LIN {X 0,Y 408.232,Z 600.263,A -85,B 0,C 180,E1 -11279.744,E2 -11279.744} C_VEL
LIN {X 0,Y 405.316,Z 581.419,A -85,B 0,C 180,E1 -11280.891,E2 -11280.891} C_VEL
LIN {X 0,Y 402.072,Z 568.541,A -85,B 0,C 180,E1 -11281.742,E2 -11281.742} C_VEL
LIN {X 0,Y 400.579,Z 563.488,A -85,B 0,C 180,E1 -11282.113,E2 -11282.113} C_VEL
LIN {X 0,Y 399.742,Z 559.755,A -85,B 0,C 180,E1 -11282.373,E2 -11282.373} C_VEL
LIN {X 0,Y 400.502,Z 548.255,A -85,B 0,C 180,E1 -11285.8,E2 -11285.8} C_VEL
LIN {X 0,Y 401.305,Z 538.061,A -85,B 0,C 180,E1 -11289.085,E2 -11289.085} C_VEL
LIN {X 0,Y 401.725,Z 533.264,A -85,B 0,C 180,E1 -11290.763,E2 -11290.763} C_VEL
LIN {X 0,Y 401.007,Z 527.558,A -85,B 0,C 180,E1 -11293.119,E2 -11293.119} C_VEL
LIN {X 0,Y 400.18,Z 522.98,A -85,B 0,C 180,E1 -11295.374,E2 -11295.374} C_VEL
LIN {X 0,Y 399.225,Z 518.76,A -85,B 0,C 180,E1 -11298.014,E2 -11298.014} C_VEL
LIN {X 0,Y 398.496,Z 515.479,A -85,B 0,C 180,E1 -11300.896,E2 -11300.896} C_VEL
LIN {X 0,Y 398.095,Z 513.82,A -85,B 0,C 180,E1 -11303.114,E2 -11303.114} C_VEL
LIN {X 0,Y 397.825,Z 512.578,A -85,B 0,C 180,E1 -11306.131,E2 -11306.131} C_VEL
LIN {X 0,Y 397.77,Z 512.409,A -85,B 0,C 180,E1 -11308.091,E2 -11308.091} C_VEL
LIN {X 0,Y 399.185,Z 514.86,A -85,B 0,C 180,E1 -11308.431,E2 -11308.431} C_VEL
LIN {X 0,Y 400.849,Z 516.713,A -85,B 0,C 180,E1 -11308.753,E2 -11308.753} C_VEL
LIN {X 0,Y 404.234,Z 521.809,A -85,B 0,C 180,E1 -11309.459,E2 -11309.459} C_VEL
LIN {X 0,Y 409.003,Z 531.362,A -85,B 0,C 180,E1 -11310.53,E2 -11310.53} C_VEL
LIN {X 0,Y 413.279,Z 542.437,A -85,B 0,C 180,E1 -11311.647,E2 -11311.647} C_VEL
LIN {X 0,Y 413.498,Z 543.353,A -85,B 0,C 180,E1 -11311.726,E2 -11311.726} C_VEL
LIN {X 0,Y 411.745,Z 560.994,A -85,B 0,C 180,E1 -11312.784,E2 -11312.784} C_VEL
LIN {X 0,Y 409.989,Z 576.551,A -85,B 0,C 180,E1 -11313.944,E2 -11313.944} C_VEL
LIN {X 0,Y 408.188,Z 591.71,A -85,B 0,C 180,E1 -11315.322,E2 -11315.322} C_VEL
LIN {X 0,Y 406.396,Z 604.533,A -85,B 0,C 180,E1 -11316.703,E2 -11316.703} C_VEL
LIN {X 0,Y 404.87,Z 615.523,A -85,B 0,C 180,E1 -11318.087,E2 -11318.087} C_VEL
LIN {X 0,Y 403.416,Z 625.962,A -85,B 0,C 180,E1 -11319.609,E2 -11319.609} C_VEL
LIN {X 0,Y 401.753,Z 636.685,A -85,B 0,C 180,E1 -11321.445,E2 -11321.445} C_VEL
LIN {X 0,Y 400.536,Z 645.216,A -85,B 0,C 180,E1 -11323.171,E2 -11323.171} C_VEL
LIN {X 0,Y 399.45,Z 652.898,A -85,B 0,C 180,E1 -11324.985,E2 -11324.985} C_VEL
LIN {X 0,Y 398.294,Z 660.864,A -85,B 0,C 180,E1 -11327.258,E2 -11327.258} C_VEL
LIN {X 0,Y 397.602,Z 666.562,A -85,B 0,C 180,E1 -11329.304,E2 -11329.304} C_VEL
LIN {X 0,Y 397.17,Z 670.116,A -85,B 0,C 180,E1 -11330.837,E2 -11330.837} C_VEL
LIN {X 0,Y 396.812,Z 673.807,A -85,B 0,C 180,E1 -11332.879,E2 -11332.879} C_VEL
LIN {X 0,Y 396.486,Z 676.537,A -85,B 0,C 180,E1 -11334.916,E2 -11334.916} C_VEL
LIN {X 0,Y 396.312,Z 678.205,A -85,B 0,C 180,E1 -11336.951,E2 -11336.951} C_VEL
LIN {X 0,Y 396.145,Z 678.944,A -85,B 0,C 180,E1 -11338.984,E2 -11338.984} C_VEL
LIN {X 0,Y 396.116,Z 678.704,A -85,B 0,C 180,E1 -11341.017,E2 -11341.017} C_VEL
LIN {X 0,Y 396.308,Z 677.478,A -85,B 0,C 180,E1 -11343.05,E2 -11343.05} C_VEL
LIN {X 0,Y 396.392,Z 675.323,A -85,B 0,C 180,E1 -11345.086,E2 -11345.086} C_VEL
LIN {X 0,Y 396.634,Z 672.104,A -85,B 0,C 180,E1 -11347.125,E2 -11347.125} C_VEL
LIN {X 0,Y 396.894,Z 667.898,A -85,B 0,C 180,E1 -11349.171,E2 -11349.171} C_VEL
LIN {X 0,Y 397.424,Z 660.965,A -85,B 0,C 180,E1 -11351.734,E2 -11351.734} C_VEL
LIN {X 0,Y 398.273,Z 653.408,A -85,B 0,C 180,E1 -11353.941,E2 -11353.941} C_VEL
LIN {X 0,Y 399.279,Z 644.403,A -85,B 0,C 180,E1 -11356.095,E2 -11356.095} C_VEL
LIN {X 0,Y 400.377,Z 635.474,A -85,B 0,C 180,E1 -11357.89,E2 -11357.89} C_VEL
LIN {X 0,Y 401.652,Z 625.081,A -85,B 0,C 180,E1 -11359.684,E2 -11359.684} C_VEL
LIN {X 0,Y 402.963,Z 614.717,A -85,B 0,C 180,E1 -11361.217,E2 -11361.217} C_VEL
LIN {X 0,Y 404.626,Z 601.75,A -85,B 0,C 180,E1 -11362.851,E2 -11362.851} C_VEL
LIN {X 0,Y 406.197,Z 588.552,A -85,B 0,C 180,E1 -11364.263,E2 -11364.263} C_VEL
LIN {X 0,Y 407.751,Z 574.631,A -85,B 0,C 180,E1 -11365.525,E2 -11365.525} C_VEL
LIN {X 0,Y 409.08,Z 561.456,A -85,B 0,C 180,E1 -11366.531,E2 -11366.531} C_VEL
LIN {X 0,Y 410.589,Z 545.552,A -85,B 0,C 180,E1 -11367.527,E2 -11367.527} C_VEL
LIN {X 0,Y 410.716,Z 541.576,A -85,B 0,C 180,E1 -11367.762,E2 -11367.762} C_VEL
LIN {X 0,Y 404.657,Z 526.643,A -85,B 0,C 180,E1 -11368.967,E2 -11368.967} C_VEL
LIN {X 0,Y 397.755,Z 511.465,A -85,B 0,C 180,E1 -11370.096,E2 -11370.096} C_VEL
LIN {X 0,Y 397.116,Z 509.333,A -85,B 0,C 180,E1 -11370.259,E2 -11370.259} C_VEL
LIN {X 0,Y 397.124,Z 509.331,A -85,B 0,C 180,E1 -11373.718,E2 -11373.718} C_VEL
LIN {X 0,Y 397.102,Z 509.334,A -85,B 0,C 180,E1 -11377.21,E2 -11377.21} C_VEL
LIN {X 0,Y 397.107,Z 509.335,A -85,B 0,C 180,E1 -11380.445,E2 -11380.445} C_VEL
LIN {X 0,Y 397.106,Z 509.333,A -85,B 0,C 180,E1 -11383.648,E2 -11383.648} C_VEL
LIN {X 0,Y 397.108,Z 509.332,A -85,B 0,C 180,E1 -11386.521,E2 -11386.521} C_VEL
LIN {X 0,Y 397.12,Z 509.334,A -85,B 0,C 180,E1 -11390.423,E2 -11390.423} C_VEL
LIN {X 0,Y 397.114,Z 509.336,A -85,B 0,C 180,E1 -11394.265,E2 -11394.265} C_VEL
LIN {X 0,Y 397.12,Z 509.336,A -85,B 0,C 180,E1 -11396.727,E2 -11396.727} C_VEL
LIN {X 0,Y 397.13,Z 509.334,A -85,B 0,C 180,E1 -11400.295,E2 -11400.295} C_VEL
LIN {X 0,Y 397.204,Z 509.363,A -85,B 0,C 180,E1 -11402.466,E2 -11402.466} C_VEL
LIN {X 0,Y 397.787,Z 513.394,A -85,B 0,C 180,E1 -11404.91,E2 -11404.91} C_VEL
LIN {X 0,Y 397.796,Z 518.959,A -85,B 0,C 180,E1 -11408.221,E2 -11408.221} C_VEL
LIN {X 0,Y 397.684,Z 524.314,A -85,B 0,C 180,E1 -11411.451,E2 -11411.451} C_VEL
LIN {X 0,Y 397.658,Z 528.743,A -85,B 0,C 180,E1 -11414.06,E2 -11414.06} C_VEL
LIN {X 0,Y 400.874,Z 536.859,A -85,B 0,C 180,E1 -11414.48,E2 -11414.48} C_VEL
LIN {X 0,Y 407.03,Z 552.39,A -85,B 0,C 180,E1 -11415.394,E2 -11415.394} C_VEL
LIN {X 0,Y 412.436,Z 568.427,A -85,B 0,C 180,E1 -11416.453,E2 -11416.453} C_VEL
LIN {X 0,Y 412.553,Z 570.388,A -85,B 0,C 180,E1 -11416.554,E2 -11416.554} C_VEL
LIN {X 0,Y 411.371,Z 585.54,A -85,B 0,C 180,E1 -11417.32,E2 -11417.32} C_VEL
LIN {X 0,Y 409.951,Z 600.302,A -85,B 0,C 180,E1 -11418.253,E2 -11418.253} C_VEL
LIN {X 0,Y 408.416,Z 614.386,A -85,B 0,C 180,E1 -11419.339,E2 -11419.339} C_VEL
LIN {X 0,Y 406.621,Z 628.646,A -85,B 0,C 180,E1 -11420.674,E2 -11420.674} C_VEL
LIN {X 0,Y 404.874,Z 641.716,A -85,B 0,C 180,E1 -11422.142,E2 -11422.142} C_VEL
LIN {X 0,Y 403.143,Z 653.798,A -85,B 0,C 180,E1 -11423.744,E2 -11423.744} C_VEL
LIN {X 0,Y 401.526,Z 664.929,A -85,B 0,C 180,E1 -11425.481,E2 -11425.481} C_VEL
LIN {X 0,Y 399.981,Z 675.704,A -85,B 0,C 180,E1 -11427.481,E2 -11427.481} C_VEL
LIN {X 0,Y 398.666,Z 684.761,A -85,B 0,C 180,E1 -11429.494,E2 -11429.494} C_VEL
LIN {X 0,Y 398.078,Z 689.301,A -85,B 0,C 180,E1 -11430.665,E2 -11430.665} C_VEL
LIN {X 0,Y 397.078,Z 692.058,A -85,B 0,C 180,E1 -11431.405,E2 -11431.405} C_VEL
LIN {X 0,Y 391.042,Z 699.537,A -85,B 0,C 180,E1 -11433.596,E2 -11433.596} C_VEL
LIN {X 0,Y 389.819,Z 701.752,A -85,B 0,C 180,E1 -11434.383,E2 -11434.383} C_VEL
LIN {X 0,Y 389.682,Z 702.392,A -85,B 0,C 180,E1 -11434.654,E2 -11434.654} C_VEL
LIN {X 0,Y 389.273,Z 706.982,A -85,B 0,C 180,E1 -11436.789,E2 -11436.789} C_VEL
LIN {X 0,Y 389,Z 709.592,A -85,B 0,C 180,E1 -11438.309,E2 -11438.309} C_VEL
LIN {X 0,Y 388.758,Z 712.241,A -85,B 0,C 180,E1 -11440.414,E2 -11440.414} C_VEL
LIN {X 0,Y 388.731,Z 713.972,A -85,B 0,C 180,E1 -11442.529,E2 -11442.529} C_VEL
LIN {X 0,Y 388.595,Z 714.684,A -85,B 0,C 180,E1 -11444.666,E2 -11444.666} C_VEL
LIN {X 0,Y 388.638,Z 714.434,A -85,B 0,C 180,E1 -11446.817,E2 -11446.817} C_VEL
LIN {X 0,Y 388.689,Z 713.166,A -85,B 0,C 180,E1 -11448.992,E2 -11448.992} C_VEL
LIN {X 0,Y 388.909,Z 710.807,A -85,B 0,C 180,E1 -11451.186,E2 -11451.186} C_VEL
LIN {X 0,Y 389.288,Z 707.379,A -85,B 0,C 180,E1 -11453.4,E2 -11453.4} C_VEL
LIN {X 0,Y 389.818,Z 702.644,A -85,B 0,C 180,E1 -11455.65,E2 -11455.65} C_VEL
LIN {X 0,Y 390.549,Z 696.64,A -85,B 0,C 180,E1 -11457.895,E2 -11457.895} C_VEL
LIN {X 0,Y 391.565,Z 689.136,A -85,B 0,C 180,E1 -11460.168,E2 -11460.168} C_VEL
LIN {X 0,Y 392.828,Z 681.236,A -85,B 0,C 180,E1 -11462.156,E2 -11462.156} C_VEL
LIN {X 0,Y 394.372,Z 671.747,A -85,B 0,C 180,E1 -11464.148,E2 -11464.148} C_VEL
LIN {X 0,Y 395.984,Z 662.193,A -85,B 0,C 180,E1 -11465.85,E2 -11465.85} C_VEL
LIN {X 0,Y 397.88,Z 650.516,A -85,B 0,C 180,E1 -11467.631,E2 -11467.631} C_VEL
LIN {X 0,Y 399.917,Z 637.964,A -85,B 0,C 180,E1 -11469.244,E2 -11469.244} C_VEL
LIN {X 0,Y 402.044,Z 623.588,A -85,B 0,C 180,E1 -11470.785,E2 -11470.785} C_VEL
LIN {X 0,Y 404.009,Z 609.267,A -85,B 0,C 180,E1 -11472.044,E2 -11472.044} C_VEL
LIN {X 0,Y 405.508,Z 596.04,A -85,B 0,C 180,E1 -11473.019,E2 -11473.019} C_VEL
LIN {X 0,Y 407.117,Z 580.483,A -85,B 0,C 180,E1 -11473.946,E2 -11473.946} C_VEL
LIN {X 0,Y 407.686,Z 571.505,A -85,B 0,C 180,E1 -11474.403,E2 -11474.403} C_VEL
LIN {X 0,Y 403.383,Z 558.004,A -85,B 0,C 180,E1 -11475.434,E2 -11475.434} C_VEL
LIN {X 0,Y 397.498,Z 543.758,A -85,B 0,C 180,E1 -11476.5,E2 -11476.5} C_VEL
LIN {X 0,Y 392.172,Z 532.891,A -85,B 0,C 180,E1 -11477.32,E2 -11477.32} C_VEL
LIN {X 0,Y 391.082,Z 530.021,A -85,B 0,C 180,E1 -11477.515,E2 -11477.515} C_VEL
LIN {X 0,Y 391.261,Z 524.474,A -85,B 0,C 180,E1 -11481.046,E2 -11481.046} C_VEL
LIN {X 0,Y 391.418,Z 519.979,A -85,B 0,C 180,E1 -11483.897,E2 -11483.897} C_VEL
LIN {X 0,Y 391.231,Z 516.544,A -85,B 0,C 180,E1 -11486.159,E2 -11486.159} C_VEL
LIN {X 0,Y 390.237,Z 511.089,A -85,B 0,C 180,E1 -11489.717,E2 -11489.717} C_VEL
LIN {X 0,Y 390.104,Z 510.207,A -85,B 0,C 180,E1 -11490.358,E2 -11490.358} C_VEL
LIN {X 0,Y 390.106,Z 510.204,A -85,B 0,C 180,E1 -11493.231,E2 -11493.231} C_VEL
LIN {X 0,Y 390.098,Z 510.204,A -85,B 0,C 180,E1 -11496.749,E2 -11496.749} C_VEL
LIN {X 0,Y 390.11,Z 510.207,A -85,B 0,C 180,E1 -11499.983,E2 -11499.983} C_VEL
LIN {X 0,Y 390.128,Z 510.198,A -85,B 0,C 180,E1 -11503.247,E2 -11503.247} C_VEL
LIN {X 0,Y 390.184,Z 510.191,A -85,B 0,C 180,E1 -11506.561,E2 -11506.561} C_VEL
LIN {X 0,Y 390.169,Z 510.193,A -85,B 0,C 180,E1 -11509.622,E2 -11509.622} C_VEL
LIN {X 0,Y 390.309,Z 510.177,A -85,B 0,C 180,E1 -11512.758,E2 -11512.758} C_VEL
LIN {X 0,Y 390.225,Z 510.185,A -85,B 0,C 180,E1 -11514.833,E2 -11514.833} C_VEL
LIN {X 0,Y 390.411,Z 510.161,A -85,B 0,C 180,E1 -11517.936,E2 -11517.936} C_VEL
LIN {X 0,Y 390.541,Z 510.151,A -85,B 0,C 180,E1 -11520,E2 -11520} C_VEL
LIN {X 0,Y 390.307,Z 510.178,A -85,B 0,C 180,E1 -11523.096,E2 -11523.096} C_VEL
LIN {X 0,Y 390.319,Z 510.172,A -85,B 0,C 180,E1 -11526.202,E2 -11526.202} C_VEL
LIN {X 0,Y 390.304,Z 510.174,A -85,B 0,C 180,E1 -11528.282,E2 -11528.282} C_VEL
LIN {X 0,Y 390.168,Z 510.187,A -85,B 0,C 180,E1 -11532.483,E2 -11532.483} C_VEL
LIN {X 0,Y 390.129,Z 510.19,A -85,B 0,C 180,E1 -11535.677,E2 -11535.677} C_VEL
LIN {X 0,Y 390.108,Z 510.177,A -85,B 0,C 180,E1 -11538.921,E2 -11538.921} C_VEL
LIN {X 0,Y 390.1,Z 510.2,A -85,B 0,C 180,E1 -11542.23,E2 -11542.23} C_VEL
LIN {X 0,Y 390.108,Z 510.179,A -85,B 0,C 180,E1 -11545.744,E2 -11545.744} C_VEL
LIN {X 0,Y 390.055,Z 510.213,A -85,B 0,C 180,E1 -11549.109,E2 -11549.109} C_VEL
LIN {X 0,Y 390.034,Z 510.214,A -85,B 0,C 180,E1 -11552.722,E2 -11552.722} C_VEL
LIN {X 0,Y 390.047,Z 510.21,A -85,B 0,C 180,E1 -11555.826,E2 -11555.826} C_VEL
LIN {X 0,Y 390.062,Z 510.224,A -85,B 0,C 180,E1 -11557.06,E2 -11557.06} C_VEL
LIN {X 0,Y 391.812,Z 517.891,A -85,B 0,C 180,E1 -11560.221,E2 -11560.221} C_VEL
LIN {X 0,Y 393.547,Z 526.096,A -85,B 0,C 180,E1 -11563.434,E2 -11563.434} C_VEL
LIN {X 0,Y 395.478,Z 535.006,A -85,B 0,C 180,E1 -11566.769,E2 -11566.769} C_VEL
LIN {X 0,Y 396.313,Z 540.139,A -85,B 0,C 180,E1 -11568.592,E2 -11568.592} C_VEL
LIN {X 0,Y 395.839,Z 547.199,A -85,B 0,C 180,E1 -11570.912,E2 -11570.912} C_VEL
LIN {X 0,Y 394.812,Z 557.025,A -85,B 0,C 180,E1 -11574.027,E2 -11574.027} C_VEL
LIN {X 0,Y 393.841,Z 567.604,A -85,B 0,C 180,E1 -11577.305,E2 -11577.305} C_VEL
LIN {X 0,Y 393.59,Z 570.386,A -85,B 0,C 180,E1 -11578.144,E2 -11578.144} C_VEL
LIN {X 0,Y 399.789,Z 593.013,A -85,B 0,C 180,E1 -11579.311,E2 -11579.311} C_VEL
LIN {X 0,Y 403.572,Z 609.943,A -85,B 0,C 180,E1 -11580.299,E2 -11580.299} C_VEL
LIN {X 0,Y 405.624,Z 620.284,A -85,B 0,C 180,E1 -11580.98,E2 -11580.98} C_VEL
LIN {X 0,Y 404.084,Z 636.161,A -85,B 0,C 180,E1 -11581.859,E2 -11581.859} C_VEL
LIN {X 0,Y 402.301,Z 650.629,A -85,B 0,C 180,E1 -11582.847,E2 -11582.847} C_VEL
LIN {X 0,Y 400.31,Z 665.785,A -85,B 0,C 180,E1 -11584.107,E2 -11584.107} C_VEL
LIN {X 0,Y 398.33,Z 679.819,A -85,B 0,C 180,E1 -11585.506,E2 -11585.506} C_VEL
LIN {X 0,Y 396.467,Z 692.875,A -85,B 0,C 180,E1 -11587.048,E2 -11587.048} C_VEL
LIN {X 0,Y 394.588,Z 705.859,A -85,B 0,C 180,E1 -11588.86,E2 -11588.86} C_VEL
LIN {X 0,Y 393.024,Z 716.9,A -85,B 0,C 180,E1 -11590.683,E2 -11590.683} C_VEL
LIN {X 0,Y 391.815,Z 726.351,A -85,B 0,C 180,E1 -11592.517,E2 -11592.517} C_VEL
LIN {X 0,Y 390.658,Z 735.563,A -85,B 0,C 180,E1 -11594.613,E2 -11594.613} C_VEL
LIN {X 0,Y 389.937,Z 743.324,A -85,B 0,C 180,E1 -11596.72,E2 -11596.72} C_VEL
LIN {X 0,Y 389.28,Z 750.35,A -85,B 0,C 180,E1 -11599.074,E2 -11599.074} C_VEL
LIN {X 0,Y 389.016,Z 755.311,A -85,B 0,C 180,E1 -11601.168,E2 -11601.168} C_VEL
LIN {X 0,Y 388.916,Z 759.796,A -85,B 0,C 180,E1 -11603.66,E2 -11603.66} C_VEL
LIN {X 0,Y 388.73,Z 762.483,A -85,B 0,C 180,E1 -11605.854,E2 -11605.854} C_VEL
LIN {X 0,Y 388.871,Z 763.909,A -85,B 0,C 180,E1 -11607.93,E2 -11607.93} C_VEL
LIN {X 0,Y 388.837,Z 764.362,A -85,B 0,C 180,E1 -11610.001,E2 -11610.001} C_VEL
LIN {X 0,Y 388.937,Z 763.726,A -85,B 0,C 180,E1 -11612.072,E2 -11612.072} C_VEL
LIN {X 0,Y 388.785,Z 762.123,A -85,B 0,C 180,E1 -11614.148,E2 -11614.148} C_VEL
LIN {X 0,Y 388.957,Z 759.368,A -85,B 0,C 180,E1 -11616.395,E2 -11616.395} C_VEL
LIN {X 0,Y 389.029,Z 754.96,A -85,B 0,C 180,E1 -11618.834,E2 -11618.834} C_VEL
LIN {X 0,Y 389.306,Z 750.025,A -85,B 0,C 180,E1 -11620.928,E2 -11620.928} C_VEL
LIN {X 0,Y 389.953,Z 743.004,A -85,B 0,C 180,E1 -11623.29,E2 -11623.29} C_VEL
LIN {X 0,Y 390.796,Z 734.274,A -85,B 0,C 180,E1 -11625.651,E2 -11625.651} C_VEL
LIN {X 0,Y 391.968,Z 724.851,A -85,B 0,C 180,E1 -11627.748,E2 -11627.748} C_VEL
LIN {X 0,Y 393.25,Z 715.147,A -85,B 0,C 180,E1 -11629.579,E2 -11629.579} C_VEL
LIN {X 0,Y 394.82,Z 703.819,A -85,B 0,C 180,E1 -11631.403,E2 -11631.403} C_VEL
LIN {X 0,Y 396.608,Z 691.46,A -85,B 0,C 180,E1 -11633.084,E2 -11633.084} C_VEL
LIN {X 0,Y 398.478,Z 677.931,A -85,B 0,C 180,E1 -11634.626,E2 -11634.626} C_VEL
LIN {X 0,Y 400.243,Z 664.612,A -85,B 0,C 180,E1 -11635.9,E2 -11635.9} C_VEL
LIN {X 0,Y 401.991,Z 650.43,A -85,B 0,C 180,E1 -11637.037,E2 -11637.037} C_VEL
LIN {X 0,Y 403.683,Z 635.143,A -85,B 0,C 180,E1 -11638.039,E2 -11638.039} C_VEL
LIN {X 0,Y 405.114,Z 620.404,A -85,B 0,C 180,E1 -11638.835,E2 -11638.835} C_VEL
LIN {X 0,Y 402.239,Z 602.925,A -85,B 0,C 180,E1 -11640.134,E2 -11640.134} C_VEL
LIN {X 0,Y 399.73,Z 584.771,A -85,B 0,C 180,E1 -11641.317,E2 -11641.317} C_VEL
LIN {X 0,Y 396.715,Z 571.614,A -85,B 0,C 180,E1 -11642.248,E2 -11642.248} C_VEL
LIN {X 0,Y 394.133,Z 562.415,A -85,B 0,C 180,E1 -11642.969,E2 -11642.969} C_VEL
LIN {X 0,Y 393.01,Z 558.534,A -85,B 0,C 180,E1 -11643.296,E2 -11643.296} C_VEL
LIN {X 0,Y 392.946,Z 557.557,A -85,B 0,C 180,E1 -11643.416,E2 -11643.416} C_VEL
LIN {X 0,Y 393.854,Z 546.412,A -85,B 0,C 180,E1 -11646.895,E2 -11646.895} C_VEL
LIN {X 0,Y 394.693,Z 537.205,A -85,B 0,C 180,E1 -11650.034,E2 -11650.034} C_VEL
LIN {X 0,Y 394.715,Z 533.136,A -85,B 0,C 180,E1 -11651.599,E2 -11651.599} C_VEL
LIN {X 0,Y 393.875,Z 527.61,A -85,B 0,C 180,E1 -11654.099,E2 -11654.099} C_VEL
LIN {X 0,Y 393.042,Z 523.275,A -85,B 0,C 180,E1 -11656.495,E2 -11656.495} C_VEL
LIN {X 0,Y 392.021,Z 518.861,A -85,B 0,C 180,E1 -11659.805,E2 -11659.805} C_VEL
LIN {X 0,Y 391.498,Z 516.574,A -85,B 0,C 180,E1 -11662.385,E2 -11662.385} C_VEL
LIN {X 0,Y 391.099,Z 514.905,A -85,B 0,C 180,E1 -11665.753,E2 -11665.753} C_VEL
LIN {X 0,Y 391.038,Z 514.772,A -85,B 0,C 180,E1 -11667.127,E2 -11667.127} C_VEL
LIN {X 0,Y 392.595,Z 517.244,A -85,B 0,C 180,E1 -11667.534,E2 -11667.534} C_VEL
LIN {X 0,Y 394.151,Z 518.801,A -85,B 0,C 180,E1 -11667.87,E2 -11667.87} C_VEL
LIN {X 0,Y 398.297,Z 524.304,A -85,B 0,C 180,E1 -11668.787,E2 -11668.787} C_VEL
LIN {X 0,Y 403.505,Z 534.578,A -85,B 0,C 180,E1 -11670.061,E2 -11670.061} C_VEL
LIN {X 0,Y 407.507,Z 545.247,A -85,B 0,C 180,E1 -11671.204,E2 -11671.204} C_VEL
LIN {X 0,Y 405.829,Z 562.036,A -85,B 0,C 180,E1 -11672.253,E2 -11672.253} C_VEL
LIN {X 0,Y 404.001,Z 576.936,A -85,B 0,C 180,E1 -11673.388,E2 -11673.388} C_VEL
LIN {X 0,Y 402.224,Z 590.843,A -85,B 0,C 180,E1 -11674.654,E2 -11674.654} C_VEL
LIN {X 0,Y 400.211,Z 604.901,A -85,B 0,C 180,E1 -11676.178,E2 -11676.178} C_VEL
LIN {X 0,Y 398.428,Z 616.898,A -85,B 0,C 180,E1 -11677.714,E2 -11677.714} C_VEL
LIN {X 0,Y 396.631,Z 628.788,A -85,B 0,C 180,E1 -11679.516,E2 -11679.516} C_VEL
LIN {X 0,Y 394.961,Z 638.951,A -85,B 0,C 180,E1 -11681.32,E2 -11681.32} C_VEL
LIN {X 0,Y 393.416,Z 648.664,A -85,B 0,C 180,E1 -11683.392,E2 -11683.392} C_VEL
LIN {X 0,Y 392.233,Z 656.733,A -85,B 0,C 180,E1 -11685.473,E2 -11685.473} C_VEL
LIN {X 0,Y 391.201,Z 663.389,A -85,B 0,C 180,E1 -11687.551,E2 -11687.551} C_VEL
LIN {X 0,Y 390.582,Z 668.818,A -85,B 0,C 180,E1 -11689.634,E2 -11689.634} C_VEL
LIN {X 0,Y 390.038,Z 673.053,A -85,B 0,C 180,E1 -11691.712,E2 -11691.712} C_VEL
LIN {X 0,Y 389.722,Z 676.204,A -85,B 0,C 180,E1 -11693.789,E2 -11693.789} C_VEL
LIN {X 0,Y 389.446,Z 678.388,A -85,B 0,C 180,E1 -11695.861,E2 -11695.861} C_VEL
LIN {X 0,Y 389.175,Z 679.546,A -85,B 0,C 180,E1 -11697.931,E2 -11697.931} C_VEL
LIN {X 0,Y 389.059,Z 679.802,A -85,B 0,C 180,E1 -11700,E2 -11700} C_VEL
LIN {X 0,Y 389.136,Z 678.995,A -85,B 0,C 180,E1 -11702.07,E2 -11702.07} C_VEL
LIN {X 0,Y 389.385,Z 677.273,A -85,B 0,C 180,E1 -11704.141,E2 -11704.141} C_VEL
LIN {X 0,Y 389.351,Z 674.549,A -85,B 0,C 180,E1 -11706.218,E2 -11706.218} C_VEL
LIN {X 0,Y 389.706,Z 670.773,A -85,B 0,C 180,E1 -11708.296,E2 -11708.296} C_VEL
LIN {X 0,Y 390.054,Z 665.928,A -85,B 0,C 180,E1 -11710.381,E2 -11710.381} C_VEL
LIN {X 0,Y 390.629,Z 659.834,A -85,B 0,C 180,E1 -11712.469,E2 -11712.469} C_VEL
LIN {X 0,Y 391.46,Z 652.448,A -85,B 0,C 180,E1 -11714.558,E2 -11714.558} C_VEL
LIN {X 0,Y 392.597,Z 643.583,A -85,B 0,C 180,E1 -11716.644,E2 -11716.644} C_VEL
LIN {X 0,Y 393.969,Z 632.977,A -85,B 0,C 180,E1 -11718.73,E2 -11718.73} C_VEL
LIN {X 0,Y 395.351,Z 621.954,A -85,B 0,C 180,E1 -11720.554,E2 -11720.554} C_VEL
LIN {X 0,Y 396.836,Z 610.953,A -85,B 0,C 180,E1 -11722.108,E2 -11722.108} C_VEL
LIN {X 0,Y 398.342,Z 599.269,A -85,B 0,C 180,E1 -11723.541,E2 -11723.541} C_VEL
LIN {X 0,Y 400.158,Z 584.503,A -85,B 0,C 180,E1 -11725.069,E2 -11725.069} C_VEL
LIN {X 0,Y 401.723,Z 571.203,A -85,B 0,C 180,E1 -11726.215,E2 -11726.215} C_VEL
LIN {X 0,Y 403.139,Z 556.268,A -85,B 0,C 180,E1 -11727.307,E2 -11727.307} C_VEL
LIN {X 0,Y 404.236,Z 543.771,A -85,B 0,C 180,E1 -11728.073,E2 -11728.073} C_VEL
LIN {X 0,Y 397.518,Z 527.206,A -85,B 0,C 180,E1 -11729.456,E2 -11729.456} C_VEL
LIN {X 0,Y 390.79,Z 512.6,A -85,B 0,C 180,E1 -11730.573,E2 -11730.573} C_VEL
LIN {X 0,Y 390.062,Z 510.212,A -85,B 0,C 180,E1 -11730.732,E2 -11730.732} C_VEL
LIN {X 0,Y 390.073,Z 510.209,A -85,B 0,C 180,E1 -11734.025,E2 -11734.025} C_VEL
LIN {X 0,Y 390.05,Z 510.214,A -85,B 0,C 180,E1 -11737.551,E2 -11737.551} C_VEL
LIN {X 0,Y 390.061,Z 510.211,A -85,B 0,C 180,E1 -11740.821,E2 -11740.821} C_VEL
LIN {X 0,Y 390.06,Z 510.21,A -85,B 0,C 180,E1 -11743.886,E2 -11743.886} C_VEL
LIN {X 0,Y 390.063,Z 510.209,A -85,B 0,C 180,E1 -11746.79,E2 -11746.79} C_VEL
LIN {X 0,Y 390.062,Z 510.21,A -85,B 0,C 180,E1 -11749.56,E2 -11749.56} C_VEL
LIN {X 0,Y 390.049,Z 510.212,A -85,B 0,C 180,E1 -11752.449,E2 -11752.449} C_VEL
LIN {X 0,Y 390.074,Z 510.214,A -85,B 0,C 180,E1 -11756.045,E2 -11756.045} C_VEL
LIN {X 0,Y 390.053,Z 510.217,A -85,B 0,C 180,E1 -11759.869,E2 -11759.869} C_VEL
LIN {X 0,Y 390.157,Z 510.377,A -85,B 0,C 180,E1 -11762.218,E2 -11762.218} C_VEL
LIN {X 0,Y 390.754,Z 514.002,A -85,B 0,C 180,E1 -11764.426,E2 -11764.426} C_VEL
LIN {X 0,Y 390.847,Z 517.77,A -85,B 0,C 180,E1 -11766.696,E2 -11766.696} C_VEL
LIN {X 0,Y 390.769,Z 523.277,A -85,B 0,C 180,E1 -11770.018,E2 -11770.018} C_VEL
LIN {X 0,Y 390.674,Z 528.948,A -85,B 0,C 180,E1 -11773.482,E2 -11773.482} C_VEL
LIN {X 0,Y 391.754,Z 532.057,A -85,B 0,C 180,E1 -11773.655,E2 -11773.655} C_VEL
LIN {X 0,Y 399.059,Z 549.937,A -85,B 0,C 180,E1 -11774.705,E2 -11774.705} C_VEL
LIN {X 0,Y 404.447,Z 565.332,A -85,B 0,C 180,E1 -11775.715,E2 -11775.715} C_VEL
LIN {X 0,Y 406.187,Z 571.314,A -85,B 0,C 180,E1 -11776.133,E2 -11776.133} C_VEL
LIN {X 0,Y 404.884,Z 587.171,A -85,B 0,C 180,E1 -11776.958,E2 -11776.958} C_VEL
LIN {X 0,Y 403.362,Z 602.056,A -85,B 0,C 180,E1 -11777.93,E2 -11777.93} C_VEL
LIN {X 0,Y 401.781,Z 615.905,A -85,B 0,C 180,E1 -11779.033,E2 -11779.033} C_VEL
LIN {X 0,Y 399.952,Z 630.054,A -85,B 0,C 180,E1 -11780.389,E2 -11780.389} C_VEL
LIN {X 0,Y 398.132,Z 642.987,A -85,B 0,C 180,E1 -11781.881,E2 -11781.881} C_VEL
LIN {X 0,Y 396.454,Z 654.101,A -85,B 0,C 180,E1 -11783.382,E2 -11783.382} C_VEL
LIN {X 0,Y 394.788,Z 665.26,A -85,B 0,C 180,E1 -11785.148,E2 -11785.148} C_VEL
LIN {X 0,Y 393.165,Z 676.055,A -85,B 0,C 180,E1 -11787.181,E2 -11787.181} C_VEL
LIN {X 0,Y 391.764,Z 685.127,A -85,B 0,C 180,E1 -11789.228,E2 -11789.228} C_VEL
LIN {X 0,Y 390.864,Z 691.831,A -85,B 0,C 180,E1 -11791.029,E2 -11791.029} C_VEL
LIN {X 0,Y 390.031,Z 698.359,A -85,B 0,C 180,E1 -11793.098,E2 -11793.098} C_VEL
LIN {X 0,Y 389.682,Z 702.392,A -85,B 0,C 180,E1 -11794.654,E2 -11794.654} C_VEL
LIN {X 0,Y 388.855,Z 704.361,A -85,B 0,C 180,E1 -11795.464,E2 -11795.464} C_VEL
LIN {X 0,Y 385.718,Z 707.32,A -85,B 0,C 180,E1 -11796.786,E2 -11796.786} C_VEL
LIN {X 0,Y 383.095,Z 709.374,A -85,B 0,C 180,E1 -11797.868,E2 -11797.868} C_VEL
LIN {X 0,Y 381.931,Z 710.719,A -85,B 0,C 180,E1 -11798.718,E2 -11798.718} C_VEL
LIN {X 0,Y 381.813,Z 711.109,A -85,B 0,C 180,E1 -11799.009,E2 -11799.009} C_VEL
LIN {X 0,Y 381.676,Z 712.948,A -85,B 0,C 180,E1 -11800.609,E2 -11800.609} C_VEL
LIN {X 0,Y 381.611,Z 714.536,A -85,B 0,C 180,E1 -11802.766,E2 -11802.766} C_VEL
LIN {X 0,Y 381.506,Z 715.177,A -85,B 0,C 180,E1 -11804.944,E2 -11804.944} C_VEL
LIN {X 0,Y 381.567,Z 714.778,A -85,B 0,C 180,E1 -11807.138,E2 -11807.138} C_VEL
LIN {X 0,Y 381.645,Z 713.429,A -85,B 0,C 180,E1 -11809.357,E2 -11809.357} C_VEL
LIN {X 0,Y 381.905,Z 710.921,A -85,B 0,C 180,E1 -11811.594,E2 -11811.594} C_VEL
LIN {X 0,Y 382.338,Z 707.326,A -85,B 0,C 180,E1 -11813.852,E2 -11813.852} C_VEL
LIN {X 0,Y 382.951,Z 702.535,A -85,B 0,C 180,E1 -11816.131,E2 -11816.131} C_VEL
LIN {X 0,Y 383.775,Z 696.205,A -85,B 0,C 180,E1 -11818.475,E2 -11818.475} C_VEL
LIN {X 0,Y 385.025,Z 688.006,A -85,B 0,C 180,E1 -11820.917,E2 -11820.917} C_VEL
LIN {X 0,Y 386.488,Z 679.215,A -85,B 0,C 180,E1 -11823.059,E2 -11823.059} C_VEL
LIN {X 0,Y 388.212,Z 669.304,A -85,B 0,C 180,E1 -11825.083,E2 -11825.083} C_VEL
LIN {X 0,Y 390.038,Z 659.373,A -85,B 0,C 180,E1 -11826.805,E2 -11826.805} C_VEL
LIN {X 0,Y 391.965,Z 647.61,A -85,B 0,C 180,E1 -11828.539,E2 -11828.539} C_VEL
LIN {X 0,Y 394.099,Z 634.952,A -85,B 0,C 180,E1 -11830.105,E2 -11830.105} C_VEL
LIN {X 0,Y 396.199,Z 621.076,A -85,B 0,C 180,E1 -11831.551,E2 -11831.551} C_VEL
LIN {X 0,Y 398.209,Z 606.559,A -85,B 0,C 180,E1 -11832.801,E2 -11832.801} C_VEL
LIN {X 0,Y 399.985,Z 591.759,A -85,B 0,C 180,E1 -11833.847,E2 -11833.847} C_VEL
LIN {X 0,Y 401.508,Z 576.128,A -85,B 0,C 180,E1 -11834.721,E2 -11834.721} C_VEL
LIN {X 0,Y 401.648,Z 574.562,A -85,B 0,C 180,E1 -11834.802,E2 -11834.802} C_VEL
LIN {X 0,Y 399.455,Z 566.295,A -85,B 0,C 180,E1 -11835.444,E2 -11835.444} C_VEL
LIN {X 0,Y 394.724,Z 553.39,A -85,B 0,C 180,E1 -11836.462,E2 -11836.462} C_VEL
LIN {X 0,Y 388.951,Z 540.503,A -85,B 0,C 180,E1 -11837.479,E2 -11837.479} C_VEL
LIN {X 0,Y 384.469,Z 531.49,A -85,B 0,C 180,E1 -11838.182,E2 -11838.182} C_VEL
LIN {X 0,Y 384.212,Z 530.464,A -85,B 0,C 180,E1 -11838.259,E2 -11838.259} C_VEL
LIN {X 0,Y 384.41,Z 524.912,A -85,B 0,C 180,E1 -11841.824,E2 -11841.824} C_VEL
LIN {X 0,Y 384.504,Z 521.219,A -85,B 0,C 180,E1 -11844.204,E2 -11844.204} C_VEL
LIN {X 0,Y 384.447,Z 519.277,A -85,B 0,C 180,E1 -11845.479,E2 -11845.479} C_VEL
LIN {X 0,Y 383.9,Z 515.687,A -85,B 0,C 180,E1 -11847.933,E2 -11847.933} C_VEL
LIN {X 0,Y 383.029,Z 511.09,A -85,B 0,C 180,E1 -11850.981,E2 -11850.981} C_VEL
LIN {X 0,Y 383.072,Z 511.083,A -85,B 0,C 180,E1 -11854.02,E2 -11854.02} C_VEL
LIN {X 0,Y 383.005,Z 511.09,A -85,B 0,C 180,E1 -11857.334,E2 -11857.334} C_VEL
LIN {X 0,Y 383.063,Z 511.08,A -85,B 0,C 180,E1 -11860.716,E2 -11860.716} C_VEL
LIN {X 0,Y 383.071,Z 511.078,A -85,B 0,C 180,E1 -11864.026,E2 -11864.026} C_VEL
LIN {X 0,Y 383.131,Z 511.075,A -85,B 0,C 180,E1 -11867.283,E2 -11867.283} C_VEL
LIN {X 0,Y 383.147,Z 511.073,A -85,B 0,C 180,E1 -11870.497,E2 -11870.497} C_VEL
LIN {X 0,Y 383.264,Z 511.053,A -85,B 0,C 180,E1 -11872.625,E2 -11872.625} C_VEL
LIN {X 0,Y 383.197,Z 511.06,A -85,B 0,C 180,E1 -11874.738,E2 -11874.738} C_VEL
LIN {X 0,Y 383.378,Z 511.037,A -85,B 0,C 180,E1 -11877.898,E2 -11877.898} C_VEL
LIN {X 0,Y 383.511,Z 511.027,A -85,B 0,C 180,E1 -11880,E2 -11880} C_VEL
LIN {X 0,Y 383.243,Z 511.058,A -85,B 0,C 180,E1 -11883.153,E2 -11883.153} C_VEL
LIN {X 0,Y 383.276,Z 511.05,A -85,B 0,C 180,E1 -11886.316,E2 -11886.316} C_VEL
LIN {X 0,Y 383.249,Z 511.051,A -85,B 0,C 180,E1 -11888.435,E2 -11888.435} C_VEL
LIN {X 0,Y 383.098,Z 511.071,A -85,B 0,C 180,E1 -11891.642,E2 -11891.642} C_VEL
LIN {X 0,Y 383.101,Z 511.075,A -85,B 0,C 180,E1 -11894.882,E2 -11894.882} C_VEL
LIN {X 0,Y 383.083,Z 511.041,A -85,B 0,C 180,E1 -11898.172,E2 -11898.172} C_VEL
LIN {X 0,Y 383.063,Z 511.082,A -85,B 0,C 180,E1 -11901.526,E2 -11901.526} C_VEL
LIN {X 0,Y 383.043,Z 511.049,A -85,B 0,C 180,E1 -11904.96,E2 -11904.96} C_VEL
LIN {X 0,Y 383.039,Z 511.085,A -85,B 0,C 180,E1 -11908.492,E2 -11908.492} C_VEL
LIN {X 0,Y 383.002,Z 511.089,A -85,B 0,C 180,E1 -11912.15,E2 -11912.15} C_VEL
LIN {X 0,Y 383.008,Z 511.087,A -85,B 0,C 180,E1 -11914.668,E2 -11914.668} C_VEL
LIN {X 0,Y 383.038,Z 511.132,A -85,B 0,C 180,E1 -11916.513,E2 -11916.513} C_VEL
LIN {X 0,Y 384.853,Z 519.24,A -85,B 0,C 180,E1 -11919.919,E2 -11919.919} C_VEL
LIN {X 0,Y 386.701,Z 527.921,A -85,B 0,C 180,E1 -11923.369,E2 -11923.369} C_VEL
LIN {X 0,Y 388.816,Z 537.742,A -85,B 0,C 180,E1 -11927.088,E2 -11927.088} C_VEL
LIN {X 0,Y 389.415,Z 542.483,A -85,B 0,C 180,E1 -11928.778,E2 -11928.778} C_VEL
LIN {X 0,Y 388.642,Z 550.81,A -85,B 0,C 180,E1 -11931.523,E2 -11931.523} C_VEL
LIN {X 0,Y 387.667,Z 560.619,A -85,B 0,C 180,E1 -11934.666,E2 -11934.666} C_VEL
LIN {X 0,Y 386.807,Z 569.997,A -85,B 0,C 180,E1 -11937.551,E2 -11937.551} C_VEL
LIN {X 0,Y 393.339,Z 593.753,A -85,B 0,C 180,E1 -11938.829,E2 -11938.829} C_VEL
LIN {X 0,Y 396.924,Z 610.361,A -85,B 0,C 180,E1 -11939.828,E2 -11939.828} C_VEL
LIN {X 0,Y 399.148,Z 621.796,A -85,B 0,C 180,E1 -11940.611,E2 -11940.611} C_VEL
LIN {X 0,Y 397.296,Z 638.989,A -85,B 0,C 180,E1 -11941.616,E2 -11941.616} C_VEL
LIN {X 0,Y 395.159,Z 654.932,A -85,B 0,C 180,E1 -11942.78,E2 -11942.78} C_VEL
LIN {X 0,Y 393.013,Z 670.376,A -85,B 0,C 180,E1 -11944.16,E2 -11944.16} C_VEL
LIN {X 0,Y 391.125,Z 683.732,A -85,B 0,C 180,E1 -11945.59,E2 -11945.59} C_VEL
LIN {X 0,Y 389.16,Z 696.344,A -85,B 0,C 180,E1 -11947.184,E2 -11947.184} C_VEL
LIN {X 0,Y 387.301,Z 708.441,A -85,B 0,C 180,E1 -11949,E2 -11949} C_VEL
LIN {X 0,Y 385.638,Z 720.05,A -85,B 0,C 180,E1 -11951.069,E2 -11951.069} C_VEL
LIN {X 0,Y 384.46,Z 729.291,A -85,B 0,C 180,E1 -11952.995,E2 -11952.995} C_VEL
LIN {X 0,Y 383.34,Z 737.904,A -85,B 0,C 180,E1 -11955.129,E2 -11955.129} C_VEL
LIN {X 0,Y 382.659,Z 745.088,A -85,B 0,C 180,E1 -11957.269,E2 -11957.269} C_VEL
LIN {X 0,Y 382.091,Z 750.979,A -85,B 0,C 180,E1 -11959.402,E2 -11959.402} C_VEL
LIN {X 0,Y 381.89,Z 755.699,A -85,B 0,C 180,E1 -11961.535,E2 -11961.535} C_VEL
LIN {X 0,Y 381.844,Z 759.255,A -85,B 0,C 180,E1 -11963.661,E2 -11963.661} C_VEL
LIN {X 0,Y 381.661,Z 761.773,A -85,B 0,C 180,E1 -11965.777,E2 -11965.777} C_VEL
LIN {X 0,Y 381.802,Z 763.188,A -85,B 0,C 180,E1 -11967.891,E2 -11967.891} C_VEL
LIN {X 0,Y 381.793,Z 763.675,A -85,B 0,C 180,E1 -11970.001,E2 -11970.001} C_VEL
LIN {X 0,Y 381.863,Z 763.145,A -85,B 0,C 180,E1 -11972.111,E2 -11972.111} C_VEL
LIN {X 0,Y 381.708,Z 761.69,A -85,B 0,C 180,E1 -11974.225,E2 -11974.225} C_VEL
LIN {X 0,Y 381.885,Z 759.066,A -85,B 0,C 180,E1 -11976.394,E2 -11976.394} C_VEL
LIN {X 0,Y 381.934,Z 754.496,A -85,B 0,C 180,E1 -11979,E2 -11979} C_VEL
LIN {X 0,Y 382.27,Z 749.561,A -85,B 0,C 180,E1 -11981.131,E2 -11981.131} C_VEL
LIN {X 0,Y 382.878,Z 743.02,A -85,B 0,C 180,E1 -11983.383,E2 -11983.383} C_VEL
LIN {X 0,Y 383.713,Z 734.831,A -85,B 0,C 180,E1 -11985.675,E2 -11985.675} C_VEL
LIN {X 0,Y 384.899,Z 725.61,A -85,B 0,C 180,E1 -11987.81,E2 -11987.81} C_VEL
LIN {X 0,Y 386.437,Z 714.617,A -85,B 0,C 180,E1 -11989.939,E2 -11989.939} C_VEL
LIN {X 0,Y 388.086,Z 703.252,A -85,B 0,C 180,E1 -11991.793,E2 -11991.793} C_VEL
LIN {X 0,Y 389.964,Z 690.88,A -85,B 0,C 180,E1 -11993.5,E2 -11993.5} C_VEL
LIN {X 0,Y 391.908,Z 677.333,A -85,B 0,C 180,E1 -11995.067,E2 -11995.067} C_VEL
LIN {X 0,Y 393.788,Z 663.969,A -85,B 0,C 180,E1 -11996.357,E2 -11996.357} C_VEL
LIN {X 0,Y 395.585,Z 649.701,A -85,B 0,C 180,E1 -11997.512,E2 -11997.512} C_VEL
LIN {X 0,Y 397.379,Z 634.32,A -85,B 0,C 180,E1 -11998.524,E2 -11998.524} C_VEL
LIN {X 0,Y 398.671,Z 622.184,A -85,B 0,C 180,E1 -11999.23,E2 -11999.23} C_VEL
LIN {X 0,Y 396.234,Z 605.191,A -85,B 0,C 180,E1 -12000.566,E2 -12000.566} C_VEL
LIN {X 0,Y 393.942,Z 586.52,A -85,B 0,C 180,E1 -12001.873,E2 -12001.873} C_VEL
LIN {X 0,Y 390.732,Z 571.653,A -85,B 0,C 180,E1 -12003.003,E2 -12003.003} C_VEL
LIN {X 0,Y 387.51,Z 560.649,A -85,B 0,C 180,E1 -12003.985,E2 -12003.985} C_VEL
LIN {X 0,Y 386.257,Z 556.104,A -85,B 0,C 180,E1 -12004.408,E2 -12004.408} C_VEL
LIN {X 0,Y 386.225,Z 555.424,A -85,B 0,C 180,E1 -12004.522,E2 -12004.522} C_VEL
LIN {X 0,Y 387.022,Z 546.395,A -85,B 0,C 180,E1 -12007.469,E2 -12007.469} C_VEL
LIN {X 0,Y 387.967,Z 537.351,A -85,B 0,C 180,E1 -12010.704,E2 -12010.704} C_VEL
LIN {X 0,Y 387.549,Z 532.442,A -85,B 0,C 180,E1 -12012.798,E2 -12012.798} C_VEL
LIN {X 0,Y 386.788,Z 527.839,A -85,B 0,C 180,E1 -12015.125,E2 -12015.125} C_VEL
LIN {X 0,Y 385.882,Z 523.863,A -85,B 0,C 180,E1 -12017.634,E2 -12017.634} C_VEL
LIN {X 0,Y 385.198,Z 520.649,A -85,B 0,C 180,E1 -12020.315,E2 -12020.315} C_VEL
LIN {X 0,Y 384.603,Z 518.154,A -85,B 0,C 180,E1 -12023.518,E2 -12023.518} C_VEL
LIN {X 0,Y 384.367,Z 517.124,A -85,B 0,C 180,E1 -12026.016,E2 -12026.016} C_VEL
LIN {X 0,Y 385.911,Z 519.589,A -85,B 0,C 180,E1 -12026.486,E2 -12026.486} C_VEL
LIN {X 0,Y 387.632,Z 521.236,A -85,B 0,C 180,E1 -12026.913,E2 -12026.913} C_VEL
LIN {X 0,Y 389.925,Z 523.96,A -85,B 0,C 180,E1 -12027.482,E2 -12027.482} C_VEL
LIN {X 0,Y 394.307,Z 530.118,A -85,B 0,C 180,E1 -12028.548,E2 -12028.548} C_VEL
LIN {X 0,Y 399.22,Z 540.739,A -85,B 0,C 180,E1 -12029.904,E2 -12029.904} C_VEL
LIN {X 0,Y 401.546,Z 547.353,A -85,B 0,C 180,E1 -12030.656,E2 -12030.656} C_VEL
LIN {X 0,Y 401.721,Z 549.089,A -85,B 0,C 180,E1 -12030.793,E2 -12030.793} C_VEL
LIN {X 0,Y 399.862,Z 564.617,A -85,B 0,C 180,E1 -12031.802,E2 -12031.802} C_VEL
LIN {X 0,Y 397.754,Z 580.646,A -85,B 0,C 180,E1 -12033.079,E2 -12033.079} C_VEL
LIN {X 0,Y 395.71,Z 595.179,A -85,B 0,C 180,E1 -12034.489,E2 -12034.489} C_VEL
LIN {X 0,Y 393.605,Z 608.68,A -85,B 0,C 180,E1 -12036.033,E2 -12036.033} C_VEL
LIN {X 0,Y 391.744,Z 620.142,A -85,B 0,C 180,E1 -12037.591,E2 -12037.591} C_VEL
LIN {X 0,Y 389.828,Z 631.659,A -85,B 0,C 180,E1 -12039.419,E2 -12039.419} C_VEL
LIN {X 0,Y 388.129,Z 641.457,A -85,B 0,C 180,E1 -12041.252,E2 -12041.252} C_VEL
LIN {X 0,Y 386.714,Z 649.855,A -85,B 0,C 180,E1 -12043.096,E2 -12043.096} C_VEL
LIN {X 0,Y 385.433,Z 657.835,A -85,B 0,C 180,E1 -12045.211,E2 -12045.211} C_VEL
LIN {X 0,Y 384.35,Z 664.467,A -85,B 0,C 180,E1 -12047.325,E2 -12047.325} C_VEL
LIN {X 0,Y 383.656,Z 669.835,A -85,B 0,C 180,E1 -12049.445,E2 -12049.445} C_VEL
LIN {X 0,Y 383.077,Z 674.028,A -85,B 0,C 180,E1 -12051.561,E2 -12051.561} C_VEL
LIN {X 0,Y 382.723,Z 677.153,A -85,B 0,C 180,E1 -12053.675,E2 -12053.675} C_VEL
LIN {X 0,Y 382.424,Z 679.305,A -85,B 0,C 180,E1 -12055.785,E2 -12055.785} C_VEL
LIN {X 0,Y 382.132,Z 680.415,A -85,B 0,C 180,E1 -12057.892,E2 -12057.892} C_VEL
LIN {X 0,Y 382.008,Z 680.629,A -85,B 0,C 180,E1 -12060,E2 -12060} C_VEL
LIN {X 0,Y 382.093,Z 679.776,A -85,B 0,C 180,E1 -12062.109,E2 -12062.109} C_VEL
LIN {X 0,Y 382.328,Z 678.013,A -85,B 0,C 180,E1 -12064.217,E2 -12064.217} C_VEL
LIN {X 0,Y 382.323,Z 675.238,A -85,B 0,C 180,E1 -12066.333,E2 -12066.333} C_VEL
LIN {X 0,Y 382.697,Z 671.41,A -85,B 0,C 180,E1 -12068.449,E2 -12068.449} C_VEL
LIN {X 0,Y 383.075,Z 666.51,A -85,B 0,C 180,E1 -12070.572,E2 -12070.572} C_VEL
LIN {X 0,Y 383.698,Z 660.34,A -85,B 0,C 180,E1 -12072.698,E2 -12072.698} C_VEL
LIN {X 0,Y 384.552,Z 652.882,A -85,B 0,C 180,E1 -12074.825,E2 -12074.825} C_VEL
LIN {X 0,Y 385.76,Z 643.922,A -85,B 0,C 180,E1 -12076.948,E2 -12076.948} C_VEL
LIN {X 0,Y 387.191,Z 633.217,A -85,B 0,C 180,E1 -12079.07,E2 -12079.07} C_VEL
LIN {X 0,Y 388.641,Z 622.124,A -85,B 0,C 180,E1 -12080.926,E2 -12080.926} C_VEL
LIN {X 0,Y 390.176,Z 611.011,A -85,B 0,C 180,E1 -12082.505,E2 -12082.505} C_VEL
LIN {X 0,Y 392.053,Z 597.154,A -85,B 0,C 180,E1 -12084.186,E2 -12084.186} C_VEL
LIN {X 0,Y 393.799,Z 582.864,A -85,B 0,C 180,E1 -12085.645,E2 -12085.645} C_VEL
LIN {X 0,Y 395.467,Z 569.523,A -85,B 0,C 180,E1 -12086.788,E2 -12086.788} C_VEL
LIN {X 0,Y 396.628,Z 557.128,A -85,B 0,C 180,E1 -12087.693,E2 -12087.693} C_VEL
LIN {X 0,Y 397.696,Z 545.879,A -85,B 0,C 180,E1 -12088.396,E2 -12088.396} C_VEL
LIN {X 0,Y 391.908,Z 531.419,A -85,B 0,C 180,E1 -12089.65,E2 -12089.65} C_VEL
LIN {X 0,Y 384.202,Z 514.226,A -85,B 0,C 180,E1 -12091.013,E2 -12091.013} C_VEL
LIN {X 0,Y 383.067,Z 511.603,A -85,B 0,C 180,E1 -12091.206,E2 -12091.206} C_VEL
LIN {X 0,Y 383.003,Z 511.091,A -85,B 0,C 180,E1 -12091.248,E2 -12091.248} C_VEL
LIN {X 0,Y 383.023,Z 511.09,A -85,B 0,C 180,E1 -12094.668,E2 -12094.668} C_VEL
LIN {X 0,Y 383.006,Z 511.089,A -85,B 0,C 180,E1 -12097.904,E2 -12097.904} C_VEL
LIN {X 0,Y 382.989,Z 511.092,A -85,B 0,C 180,E1 -12101.347,E2 -12101.347} C_VEL
LIN {X 0,Y 383.001,Z 511.091,A -85,B 0,C 180,E1 -12104.303,E2 -12104.303} C_VEL
LIN {X 0,Y 383.016,Z 511.088,A -85,B 0,C 180,E1 -12107.24,E2 -12107.24} C_VEL
LIN {X 0,Y 383.021,Z 511.09,A -85,B 0,C 180,E1 -12110.413,E2 -12110.413} C_VEL
LIN {X 0,Y 383.031,Z 511.09,A -85,B 0,C 180,E1 -12114.044,E2 -12114.044} C_VEL
LIN {X 0,Y 382.993,Z 511.095,A -85,B 0,C 180,E1 -12117.578,E2 -12117.578} C_VEL
LIN {X 0,Y 382.998,Z 511.094,A -85,B 0,C 180,E1 -12120.3,E2 -12120.3} C_VEL
LIN {X 0,Y 383.08,Z 511.224,A -85,B 0,C 180,E1 -12121.831,E2 -12121.831} C_VEL
LIN {X 0,Y 383.66,Z 514.604,A -85,B 0,C 180,E1 -12123.918,E2 -12123.918} C_VEL
LIN {X 0,Y 383.871,Z 518.447,A -85,B 0,C 180,E1 -12126.266,E2 -12126.266} C_VEL
LIN {X 0,Y 383.803,Z 524.004,A -85,B 0,C 180,E1 -12129.639,E2 -12129.639} C_VEL
LIN {X 0,Y 383.701,Z 529.37,A -85,B 0,C 180,E1 -12132.924,E2 -12132.924} C_VEL
LIN {X 0,Y 384.837,Z 532.471,A -85,B 0,C 180,E1 -12133.093,E2 -12133.093} C_VEL
LIN {X 0,Y 392.306,Z 550.725,A -85,B 0,C 180,E1 -12134.196,E2 -12134.196} C_VEL
LIN {X 0,Y 397.668,Z 565.934,A -85,B 0,C 180,E1 -12135.228,E2 -12135.228} C_VEL
LIN {X 0,Y 399.771,Z 573.286,A -85,B 0,C 180,E1 -12135.751,E2 -12135.751} C_VEL
LIN {X 0,Y 398.442,Z 588.736,A -85,B 0,C 180,E1 -12136.584,E2 -12136.584} C_VEL
LIN {X 0,Y 396.806,Z 603.789,A -85,B 0,C 180,E1 -12137.598,E2 -12137.598} C_VEL
LIN {X 0,Y 394.985,Z 618.765,A -85,B 0,C 180,E1 -12138.842,E2 -12138.842} C_VEL
LIN {X 0,Y 393.082,Z 632.525,A -85,B 0,C 180,E1 -12140.22,E2 -12140.22} C_VEL
LIN {X 0,Y 391.255,Z 645.237,A -85,B 0,C 180,E1 -12141.737,E2 -12141.737} C_VEL
LIN {X 0,Y 389.18,Z 658.279,A -85,B 0,C 180,E1 -12143.594,E2 -12143.594} C_VEL
LIN {X 0,Y 387.37,Z 669.839,A -85,B 0,C 180,E1 -12145.577,E2 -12145.577} C_VEL
LIN {X 0,Y 385.721,Z 679.963,A -85,B 0,C 180,E1 -12147.649,E2 -12147.649} C_VEL
LIN {X 0,Y 384.607,Z 687.5,A -85,B 0,C 180,E1 -12149.475,E2 -12149.475} C_VEL
LIN {X 0,Y 383.608,Z 694.829,A -85,B 0,C 180,E1 -12151.574,E2 -12151.574} C_VEL
LIN {X 0,Y 382.736,Z 702.188,A -85,B 0,C 180,E1 -12154.211,E2 -12154.211} C_VEL
LIN {X 0,Y 382.197,Z 707.671,A -85,B 0,C 180,E1 -12156.791,E2 -12156.791} C_VEL
LIN {X 0,Y 381.813,Z 711.109,A -85,B 0,C 180,E1 -12159.009,E2 -12159.009} C_VEL
LIN {X 0,Y 381.064,Z 712.247,A -85,B 0,C 180,E1 -12159.873,E2 -12159.873} C_VEL
LIN {X 0,Y 378.105,Z 713.793,A -85,B 0,C 180,E1 -12161.283,E2 -12161.283} C_VEL
LIN {X 0,Y 375.625,Z 714.773,A -85,B 0,C 180,E1 -12162.429,E2 -12162.429} C_VEL
LIN {X 0,Y 374.543,Z 715.234,A -85,B 0,C 180,E1 -12163.32,E2 -12163.32} C_VEL
LIN {X 0,Y 374.444,Z 715.317,A -85,B 0,C 180,E1 -12163.622,E2 -12163.622} C_VEL
LIN {X 0,Y 374.416,Z 715.657,A -85,B 0,C 180,E1 -12165.234,E2 -12165.234} C_VEL
LIN {X 0,Y 374.487,Z 715.125,A -85,B 0,C 180,E1 -12167.473,E2 -12167.473} C_VEL
LIN {X 0,Y 374.586,Z 713.63,A -85,B 0,C 180,E1 -12169.736,E2 -12169.736} C_VEL
LIN {X 0,Y 374.893,Z 711.042,A -85,B 0,C 180,E1 -12172.019,E2 -12172.019} C_VEL
LIN {X 0,Y 375.375,Z 707.287,A -85,B 0,C 180,E1 -12174.323,E2 -12174.323} C_VEL
LIN {X 0,Y 376.082,Z 702.338,A -85,B 0,C 180,E1 -12176.646,E2 -12176.646} C_VEL
LIN {X 0,Y 376.96,Z 696.022,A -85,B 0,C 180,E1 -12178.994,E2 -12178.994} C_VEL
LIN {X 0,Y 378.276,Z 688.135,A -85,B 0,C 180,E1 -12181.345,E2 -12181.345} C_VEL
LIN {X 0,Y 379.734,Z 679.909,A -85,B 0,C 180,E1 -12183.381,E2 -12183.381} C_VEL
LIN {X 0,Y 381.59,Z 669.938,A -85,B 0,C 180,E1 -12185.46,E2 -12185.46} C_VEL
LIN {X 0,Y 383.472,Z 660.02,A -85,B 0,C 180,E1 -12187.212,E2 -12187.212} C_VEL
LIN {X 0,Y 385.508,Z 648.294,A -85,B 0,C 180,E1 -12188.971,E2 -12188.971} C_VEL
LIN {X 0,Y 387.784,Z 635.505,A -85,B 0,C 180,E1 -12190.58,E2 -12190.58} C_VEL
LIN {X 0,Y 389.941,Z 621.87,A -85,B 0,C 180,E1 -12192.027,E2 -12192.027} C_VEL
LIN {X 0,Y 392.048,Z 607.52,A -85,B 0,C 180,E1 -12193.287,E2 -12193.287} C_VEL
LIN {X 0,Y 393.871,Z 592.901,A -85,B 0,C 180,E1 -12194.339,E2 -12194.339} C_VEL
LIN {X 0,Y 395.444,Z 577.524,A -85,B 0,C 180,E1 -12195.222,E2 -12195.222} C_VEL
LIN {X 0,Y 395.57,Z 576.254,A -85,B 0,C 180,E1 -12195.287,E2 -12195.287} C_VEL
LIN {X 0,Y 392.195,Z 564.68,A -85,B 0,C 180,E1 -12196.244,E2 -12196.244} C_VEL
LIN {X 0,Y 386.804,Z 550.942,A -85,B 0,C 180,E1 -12197.384,E2 -12197.384} C_VEL
LIN {X 0,Y 380.709,Z 538.088,A -85,B 0,C 180,E1 -12198.45,E2 -12198.45} C_VEL
LIN {X 0,Y 378.389,Z 533.697,A -85,B 0,C 180,E1 -12198.822,E2 -12198.822} C_VEL
LIN {X 0,Y 377.326,Z 530.953,A -85,B 0,C 180,E1 -12199.03,E2 -12199.03} C_VEL
LIN {X 0,Y 377.516,Z 526.229,A -85,B 0,C 180,E1 -12202.095,E2 -12202.095} C_VEL
LIN {X 0,Y 377.566,Z 521.81,A -85,B 0,C 180,E1 -12204.983,E2 -12204.983} C_VEL
LIN {X 0,Y 377.184,Z 518.453,A -85,B 0,C 180,E1 -12207.292,E2 -12207.292} C_VEL
LIN {X 0,Y 376.187,Z 512.972,A -85,B 0,C 180,E1 -12210.939,E2 -12210.939} C_VEL
LIN {X 0,Y 376.026,Z 511.958,A -85,B 0,C 180,E1 -12211.792,E2 -12211.792} C_VEL
LIN {X 0,Y 375.998,Z 511.962,A -85,B 0,C 180,E1 -12214.538,E2 -12214.538} C_VEL
LIN {X 0,Y 375.963,Z 511.969,A -85,B 0,C 180,E1 -12218.045,E2 -12218.045} C_VEL
LIN {X 0,Y 376.02,Z 511.957,A -85,B 0,C 180,E1 -12221.473,E2 -12221.473} C_VEL
LIN {X 0,Y 376.05,Z 511.957,A -85,B 0,C 180,E1 -12224.832,E2 -12224.832} C_VEL
LIN {X 0,Y 376.049,Z 511.955,A -85,B 0,C 180,E1 -12228.136,E2 -12228.136} C_VEL
LIN {X 0,Y 376.247,Z 511.924,A -85,B 0,C 180,E1 -12231.876,E2 -12231.876} C_VEL
LIN {X 0,Y 376.169,Z 511.936,A -85,B 0,C 180,E1 -12234.639,E2 -12234.639} C_VEL
LIN {X 0,Y 376.344,Z 511.913,A -85,B 0,C 180,E1 -12237.859,E2 -12237.859} C_VEL
LIN {X 0,Y 376.48,Z 511.903,A -85,B 0,C 180,E1 -12240,E2 -12240} C_VEL
LIN {X 0,Y 376.182,Z 511.938,A -85,B 0,C 180,E1 -12243.212,E2 -12243.212} C_VEL
LIN {X 0,Y 376.236,Z 511.928,A -85,B 0,C 180,E1 -12246.435,E2 -12246.435} C_VEL
LIN {X 0,Y 376.195,Z 511.928,A -85,B 0,C 180,E1 -12248.595,E2 -12248.595} C_VEL
LIN {X 0,Y 376.049,Z 511.947,A -85,B 0,C 180,E1 -12251.863,E2 -12251.863} C_VEL
LIN {X 0,Y 376.048,Z 511.95,A -85,B 0,C 180,E1 -12255.167,E2 -12255.167} C_VEL
LIN {X 0,Y 376.02,Z 511.923,A -85,B 0,C 180,E1 -12258.526,E2 -12258.526} C_VEL
LIN {X 0,Y 376.012,Z 511.958,A -85,B 0,C 180,E1 -12261.951,E2 -12261.951} C_VEL
LIN {X 0,Y 375.996,Z 511.93,A -85,B 0,C 180,E1 -12265.461,E2 -12265.461} C_VEL
LIN {X 0,Y 375.966,Z 511.968,A -85,B 0,C 180,E1 -12269.079,E2 -12269.079} C_VEL
LIN {X 0,Y 375.941,Z 511.969,A -85,B 0,C 180,E1 -12272.829,E2 -12272.829} C_VEL
LIN {X 0,Y 376,Z 512.156,A -85,B 0,C 180,E1 -12276.008,E2 -12276.008} C_VEL
LIN {X 0,Y 378.018,Z 521.074,A -85,B 0,C 180,E1 -12279.819,E2 -12279.819} C_VEL
LIN {X 0,Y 379.798,Z 529.473,A -85,B 0,C 180,E1 -12283.209,E2 -12283.209} C_VEL
LIN {X 0,Y 381.646,Z 538.072,A -85,B 0,C 180,E1 -12286.524,E2 -12286.524} C_VEL
LIN {X 0,Y 382.496,Z 543.717,A -85,B 0,C 180,E1 -12288.59,E2 -12288.59} C_VEL
LIN {X 0,Y 381.79,Z 551.667,A -85,B 0,C 180,E1 -12291.256,E2 -12291.256} C_VEL
LIN {X 0,Y 380.675,Z 562.199,A -85,B 0,C 180,E1 -12294.69,E2 -12294.69} C_VEL
LIN {X 0,Y 379.937,Z 569.158,A -85,B 0,C 180,E1 -12296.907,E2 -12296.907} C_VEL
LIN {X 0,Y 386.483,Z 592.873,A -85,B 0,C 180,E1 -12298.224,E2 -12298.224} C_VEL
LIN {X 0,Y 390.277,Z 610.49,A -85,B 0,C 180,E1 -12299.324,E2 -12299.324} C_VEL
LIN {X 0,Y 392.56,Z 622.492,A -85,B 0,C 180,E1 -12300.173,E2 -12300.173} C_VEL
LIN {X 0,Y 391.005,Z 638.519,A -85,B 0,C 180,E1 -12301.116,E2 -12301.116} C_VEL
LIN {X 0,Y 389.009,Z 653.453,A -85,B 0,C 180,E1 -12302.192,E2 -12302.192} C_VEL
LIN {X 0,Y 387.012,Z 667.646,A -85,B 0,C 180,E1 -12303.439,E2 -12303.439} C_VEL
LIN {X 0,Y 384.908,Z 681.251,A -85,B 0,C 180,E1 -12304.881,E2 -12304.881} C_VEL
LIN {X 0,Y 382.91,Z 693.748,A -85,B 0,C 180,E1 -12306.45,E2 -12306.45} C_VEL
LIN {X 0,Y 380.846,Z 706.492,A -85,B 0,C 180,E1 -12308.343,E2 -12308.343} C_VEL
LIN {X 0,Y 379.156,Z 717.241,A -85,B 0,C 180,E1 -12310.229,E2 -12310.229} C_VEL
LIN {X 0,Y 377.682,Z 727.664,A -85,B 0,C 180,E1 -12312.401,E2 -12312.401} C_VEL
LIN {X 0,Y 376.478,Z 736.378,A -85,B 0,C 180,E1 -12314.574,E2 -12314.574} C_VEL
LIN {X 0,Y 375.623,Z 744.494,A -85,B 0,C 180,E1 -12317.026,E2 -12317.026} C_VEL
LIN {X 0,Y 375.055,Z 750.37,A -85,B 0,C 180,E1 -12319.201,E2 -12319.201} C_VEL
LIN {X 0,Y 374.805,Z 755.064,A -85,B 0,C 180,E1 -12321.374,E2 -12321.374} C_VEL
LIN {X 0,Y 374.756,Z 758.828,A -85,B 0,C 180,E1 -12323.683,E2 -12323.683} C_VEL
LIN {X 0,Y 374.592,Z 761.189,A -85,B 0,C 180,E1 -12325.697,E2 -12325.697} C_VEL
LIN {X 0,Y 374.736,Z 762.673,A -85,B 0,C 180,E1 -12327.852,E2 -12327.852} C_VEL
LIN {X 0,Y 374.719,Z 763.225,A -85,B 0,C 180,E1 -12330.001,E2 -12330.001} C_VEL
LIN {X 0,Y 374.789,Z 762.695,A -85,B 0,C 180,E1 -12332.15,E2 -12332.15} C_VEL
LIN {X 0,Y 374.634,Z 761.236,A -85,B 0,C 180,E1 -12334.305,E2 -12334.305} C_VEL
LIN {X 0,Y 374.784,Z 758.685,A -85,B 0,C 180,E1 -12336.461,E2 -12336.461} C_VEL
LIN {X 0,Y 374.823,Z 755.13,A -85,B 0,C 180,E1 -12338.628,E2 -12338.628} C_VEL
LIN {X 0,Y 375.078,Z 750.423,A -85,B 0,C 180,E1 -12340.801,E2 -12340.801} C_VEL
LIN {X 0,Y 375.654,Z 744.542,A -85,B 0,C 180,E1 -12342.975,E2 -12342.975} C_VEL
LIN {X 0,Y 376.392,Z 737.407,A -85,B 0,C 180,E1 -12345.155,E2 -12345.155} C_VEL
LIN {X 0,Y 377.55,Z 728.762,A -85,B 0,C 180,E1 -12347.329,E2 -12347.329} C_VEL
LIN {X 0,Y 378.764,Z 719.795,A -85,B 0,C 180,E1 -12349.235,E2 -12349.235} C_VEL
LIN {X 0,Y 380.361,Z 709.435,A -85,B 0,C 180,E1 -12351.12,E2 -12351.12} C_VEL
LIN {X 0,Y 382.176,Z 697.8,A -85,B 0,C 180,E1 -12352.915,E2 -12352.915} C_VEL
LIN {X 0,Y 384.169,Z 684.83,A -85,B 0,C 180,E1 -12354.595,E2 -12354.595} C_VEL
LIN {X 0,Y 386.124,Z 671.512,A -85,B 0,C 180,E1 -12356.048,E2 -12356.048} C_VEL
LIN {X 0,Y 388.06,Z 657.371,A -85,B 0,C 180,E1 -12357.341,E2 -12357.341} C_VEL
LIN {X 0,Y 389.861,Z 643.54,A -85,B 0,C 180,E1 -12358.39,E2 -12358.39} C_VEL
LIN {X 0,Y 392.349,Z 623.006,A -85,B 0,C 180,E1 -12359.709,E2 -12359.709} C_VEL
LIN {X 0,Y 390.274,Z 607.359,A -85,B 0,C 180,E1 -12361.028,E2 -12361.028} C_VEL
LIN {X 0,Y 388.343,Z 589.066,A -85,B 0,C 180,E1 -12362.39,E2 -12362.39} C_VEL
LIN {X 0,Y 385.452,Z 574.517,A -85,B 0,C 180,E1 -12363.585,E2 -12363.585} C_VEL
LIN {X 0,Y 382.631,Z 564.203,A -85,B 0,C 180,E1 -12364.56,E2 -12364.56} C_VEL
LIN {X 0,Y 381.166,Z 559.108,A -85,B 0,C 180,E1 -12365.081,E2 -12365.081} C_VEL
LIN {X 0,Y 379.687,Z 554.324,A -85,B 0,C 180,E1 -12365.625,E2 -12365.625} C_VEL
LIN {X 0,Y 379.569,Z 553.226,A -85,B 0,C 180,E1 -12365.744,E2 -12365.744} C_VEL
LIN {X 0,Y 380.517,Z 544.12,A -85,B 0,C 180,E1 -12368.901,E2 -12368.901} C_VEL
LIN {X 0,Y 381.128,Z 538.881,A -85,B 0,C 180,E1 -12370.884,E2 -12370.884} C_VEL
LIN {X 0,Y 380.672,Z 533.938,A -85,B 0,C 180,E1 -12373.087,E2 -12373.087} C_VEL
LIN {X 0,Y 379.967,Z 529.661,A -85,B 0,C 180,E1 -12375.344,E2 -12375.344} C_VEL
LIN {X 0,Y 379.094,Z 525.832,A -85,B 0,C 180,E1 -12377.865,E2 -12377.865} C_VEL
LIN {X 0,Y 378.367,Z 522.465,A -85,B 0,C 180,E1 -12380.837,E2 -12380.837} C_VEL
LIN {X 0,Y 377.799,Z 520.112,A -85,B 0,C 180,E1 -12384.128,E2 -12384.128} C_VEL
LIN {X 0,Y 377.741,Z 519.867,A -85,B 0,C 180,E1 -12384.721,E2 -12384.721} C_VEL
LIN {X 0,Y 379.164,Z 522.162,A -85,B 0,C 180,E1 -12385.251,E2 -12385.251} C_VEL
LIN {X 0,Y 381.202,Z 523.763,A -85,B 0,C 180,E1 -12385.816,E2 -12385.816} C_VEL
LIN {X 0,Y 383.527,Z 526.513,A -85,B 0,C 180,E1 -12386.488,E2 -12386.488} C_VEL
LIN {X 0,Y 388.901,Z 533.509,A -85,B 0,C 180,E1 -12387.93,E2 -12387.93} C_VEL
LIN {X 0,Y 391.556,Z 538.661,A -85,B 0,C 180,E1 -12388.696,E2 -12388.696} C_VEL
LIN {X 0,Y 395.139,Z 547.738,A -85,B 0,C 180,E1 -12389.868,E2 -12389.868} C_VEL
LIN {X 0,Y 396.084,Z 550.781,A -85,B 0,C 180,E1 -12390.21,E2 -12390.21} C_VEL
LIN {X 0,Y 393.936,Z 567.476,A -85,B 0,C 180,E1 -12391.35,E2 -12391.35} C_VEL
LIN {X 0,Y 391.739,Z 582.917,A -85,B 0,C 180,E1 -12392.631,E2 -12392.631} C_VEL
LIN {X 0,Y 389.353,Z 598.336,A -85,B 0,C 180,E1 -12394.185,E2 -12394.185} C_VEL
LIN {X 0,Y 387.323,Z 610.384,A -85,B 0,C 180,E1 -12395.62,E2 -12395.62} C_VEL
LIN {X 0,Y 385.365,Z 621.717,A -85,B 0,C 180,E1 -12397.199,E2 -12397.199} C_VEL
LIN {X 0,Y 383.34,Z 633.048,A -85,B 0,C 180,E1 -12399.054,E2 -12399.054} C_VEL
LIN {X 0,Y 381.516,Z 642.779,A -85,B 0,C 180,E1 -12400.915,E2 -12400.915} C_VEL
LIN {X 0,Y 379.815,Z 652.13,A -85,B 0,C 180,E1 -12403.057,E2 -12403.057} C_VEL
LIN {X 0,Y 378.652,Z 659.016,A -85,B 0,C 180,E1 -12404.939,E2 -12404.939} C_VEL
LIN {X 0,Y 377.498,Z 665.554,A -85,B 0,C 180,E1 -12407.091,E2 -12407.091} C_VEL
LIN {X 0,Y 376.735,Z 670.884,A -85,B 0,C 180,E1 -12409.249,E2 -12409.249} C_VEL
LIN {X 0,Y 376.122,Z 675.042,A -85,B 0,C 180,E1 -12411.403,E2 -12411.403} C_VEL
LIN {X 0,Y 375.728,Z 678.103,A -85,B 0,C 180,E1 -12413.557,E2 -12413.557} C_VEL
LIN {X 0,Y 375.403,Z 680.224,A -85,B 0,C 180,E1 -12415.706,E2 -12415.706} C_VEL
LIN {X 0,Y 375.091,Z 681.295,A -85,B 0,C 180,E1 -12417.853,E2 -12417.853} C_VEL
LIN {X 0,Y 374.957,Z 681.458,A -85,B 0,C 180,E1 -12420,E2 -12420} C_VEL
LIN {X 0,Y 375.051,Z 680.569,A -85,B 0,C 180,E1 -12422.148,E2 -12422.148} C_VEL
LIN {X 0,Y 375.275,Z 678.742,A -85,B 0,C 180,E1 -12424.297,E2 -12424.297} C_VEL
LIN {X 0,Y 375.298,Z 675.927,A -85,B 0,C 180,E1 -12426.452,E2 -12426.452} C_VEL
LIN {X 0,Y 375.685,Z 672.027,A -85,B 0,C 180,E1 -12428.608,E2 -12428.608} C_VEL
LIN {X 0,Y 376.099,Z 667.081,A -85,B 0,C 180,E1 -12430.77,E2 -12430.77} C_VEL
LIN {X 0,Y 376.771,Z 660.839,A -85,B 0,C 180,E1 -12432.935,E2 -12432.935} C_VEL
LIN {X 0,Y 377.653,Z 653.294,A -85,B 0,C 180,E1 -12435.102,E2 -12435.102} C_VEL
LIN {X 0,Y 378.91,Z 644.247,A -85,B 0,C 180,E1 -12437.264,E2 -12437.264} C_VEL
LIN {X 0,Y 380.216,Z 634.918,A -85,B 0,C 180,E1 -12439.154,E2 -12439.154} C_VEL
LIN {X 0,Y 381.7,Z 623.938,A -85,B 0,C 180,E1 -12441.042,E2 -12441.042} C_VEL
LIN {X 0,Y 383.565,Z 611.042,A -85,B 0,C 180,E1 -12442.915,E2 -12442.915} C_VEL
LIN {X 0,Y 385.386,Z 597.958,A -85,B 0,C 180,E1 -12444.521,E2 -12444.521} C_VEL
LIN {X 0,Y 387.163,Z 584.014,A -85,B 0,C 180,E1 -12445.972,E2 -12445.972} C_VEL
LIN {X 0,Y 389.008,Z 569.472,A -85,B 0,C 180,E1 -12447.236,E2 -12447.236} C_VEL
LIN {X 0,Y 390.168,Z 557.61,A -85,B 0,C 180,E1 -12448.112,E2 -12448.112} C_VEL
LIN {X 0,Y 391.075,Z 549.234,A -85,B 0,C 180,E1 -12448.646,E2 -12448.646} C_VEL
LIN {X 0,Y 390.897,Z 547.324,A -85,B 0,C 180,E1 -12448.787,E2 -12448.787} C_VEL
LIN {X 0,Y 384.966,Z 532.514,A -85,B 0,C 180,E1 -12450.105,E2 -12450.105} C_VEL
LIN {X 0,Y 377.303,Z 515.393,A -85,B 0,C 180,E1 -12451.515,E2 -12451.515} C_VEL
LIN {X 0,Y 376.032,Z 512.315,A -85,B 0,C 180,E1 -12451.744,E2 -12451.744} C_VEL
LIN {X 0,Y 375.977,Z 511.966,A -85,B 0,C 180,E1 -12451.797,E2 -12451.797} C_VEL
LIN {X 0,Y 375.963,Z 511.966,A -85,B 0,C 180,E1 -12455.415,E2 -12455.415} C_VEL
LIN {X 0,Y 375.98,Z 511.964,A -85,B 0,C 180,E1 -12458.271,E2 -12458.271} C_VEL
LIN {X 0,Y 375.94,Z 511.97,A -85,B 0,C 180,E1 -12461.601,E2 -12461.601} C_VEL
LIN {X 0,Y 375.932,Z 511.969,A -85,B 0,C 180,E1 -12465.269,E2 -12465.269} C_VEL
LIN {X 0,Y 375.94,Z 511.969,A -85,B 0,C 180,E1 -12468.399,E2 -12468.399} C_VEL
LIN {X 0,Y 375.98,Z 511.968,A -85,B 0,C 180,E1 -12471.729,E2 -12471.729} C_VEL
LIN {X 0,Y 375.986,Z 511.965,A -85,B 0,C 180,E1 -12475.332,E2 -12475.332} C_VEL
LIN {X 0,Y 375.964,Z 511.973,A -85,B 0,C 180,E1 -12478.438,E2 -12478.438} C_VEL
LIN {X 0,Y 376.018,Z 512.126,A -85,B 0,C 180,E1 -12481.458,E2 -12481.458} C_VEL
LIN {X 0,Y 376.636,Z 515.529,A -85,B 0,C 180,E1 -12483.597,E2 -12483.597} C_VEL
LIN {X 0,Y 376.899,Z 519.479,A -85,B 0,C 180,E1 -12486.023,E2 -12486.023} C_VEL
LIN {X 0,Y 376.843,Z 524.753,A -85,B 0,C 180,E1 -12489.246,E2 -12489.246} C_VEL
LIN {X 0,Y 376.799,Z 529.768,A -85,B 0,C 180,E1 -12492.333,E2 -12492.333} C_VEL
LIN {X 0,Y 378.066,Z 533.154,A -85,B 0,C 180,E1 -12492.528,E2 -12492.528} C_VEL
LIN {X 0,Y 385.367,Z 551.098,A -85,B 0,C 180,E1 -12493.644,E2 -12493.644} C_VEL
LIN {X 0,Y 390.596,Z 565.739,A -85,B 0,C 180,E1 -12494.659,E2 -12494.659} C_VEL
LIN {X 0,Y 393.37,Z 575.009,A -85,B 0,C 180,E1 -12495.355,E2 -12495.355} C_VEL
LIN {X 0,Y 391.976,Z 590.237,A -85,B 0,C 180,E1 -12496.195,E2 -12496.195} C_VEL
LIN {X 0,Y 390.237,Z 605.462,A -85,B 0,C 180,E1 -12497.254,E2 -12497.254} C_VEL
LIN {X 0,Y 388.352,Z 620.218,A -85,B 0,C 180,E1 -12498.517,E2 -12498.517} C_VEL
LIN {X 0,Y 386.393,Z 633.818,A -85,B 0,C 180,E1 -12499.916,E2 -12499.916} C_VEL
LIN {X 0,Y 384.645,Z 645.466,A -85,B 0,C 180,E1 -12501.329,E2 -12501.329} C_VEL
LIN {X 0,Y 382.592,Z 658.045,A -85,B 0,C 180,E1 -12503.141,E2 -12503.141} C_VEL
LIN {X 0,Y 380.837,Z 668.708,A -85,B 0,C 180,E1 -12504.97,E2 -12504.97} C_VEL
LIN {X 0,Y 379.094,Z 679.095,A -85,B 0,C 180,E1 -12507.077,E2 -12507.077} C_VEL
LIN {X 0,Y 377.853,Z 686.875,A -85,B 0,C 180,E1 -12508.933,E2 -12508.933} C_VEL
LIN {X 0,Y 376.767,Z 694.315,A -85,B 0,C 180,E1 -12511.068,E2 -12511.068} C_VEL
LIN {X 0,Y 375.882,Z 700.519,A -85,B 0,C 180,E1 -12513.214,E2 -12513.214} C_VEL
LIN {X 0,Y 375.35,Z 705.61,A -85,B 0,C 180,E1 -12515.371,E2 -12515.371} C_VEL
LIN {X 0,Y 374.967,Z 709.544,A -85,B 0,C 180,E1 -12517.538,E2 -12517.538} C_VEL
LIN {X 0,Y 374.671,Z 712.537,A -85,B 0,C 180,E1 -12519.718,E2 -12519.718} C_VEL
LIN {X 0,Y 374.563,Z 714.487,A -85,B 0,C 180,E1 -12521.91,E2 -12521.91} C_VEL
LIN {X 0,Y 374.444,Z 715.317,A -85,B 0,C 180,E1 -12523.622,E2 -12523.622} C_VEL
LIN {X 0,Y 373.749,Z 715.609,A -85,B 0,C 180,E1 -12524.52,E2 -12524.52} C_VEL
LIN {X 0,Y 370.897,Z 715.81,A -85,B 0,C 180,E1 -12525.982,E2 -12525.982} C_VEL
LIN {X 0,Y 368.51,Z 715.663,A -85,B 0,C 180,E1 -12527.163,E2 -12527.163} C_VEL
LIN {X 0,Y 367.442,Z 715.285,A -85,B 0,C 180,E1 -12528.228,E2 -12528.228} C_VEL
LIN {X 0,Y 367.423,Z 715.134,A -85,B 0,C 180,E1 -12528.382,E2 -12528.382} C_VEL
LIN {X 0,Y 367.593,Z 713.5,A -85,B 0,C 180,E1 -12530.473,E2 -12530.473} C_VEL
LIN {X 0,Y 367.898,Z 711.162,A -85,B 0,C 180,E1 -12532.46,E2 -12532.46} C_VEL
LIN {X 0,Y 368.448,Z 707.25,A -85,B 0,C 180,E1 -12534.81,E2 -12534.81} C_VEL
LIN {X 0,Y 369.222,Z 702.133,A -85,B 0,C 180,E1 -12537.181,E2 -12537.181} C_VEL
LIN {X 0,Y 370.228,Z 695.667,A -85,B 0,C 180,E1 -12539.573,E2 -12539.573} C_VEL
LIN {X 0,Y 371.694,Z 687.654,A -85,B 0,C 180,E1 -12541.965,E2 -12541.965} C_VEL
LIN {X 0,Y 373.285,Z 679.107,A -85,B 0,C 180,E1 -12544.064,E2 -12544.064} C_VEL
LIN {X 0,Y 375.14,Z 669.588,A -85,B 0,C 180,E1 -12546.04,E2 -12546.04} C_VEL
LIN {X 0,Y 377.267,Z 658.856,A -85,B 0,C 180,E1 -12547.932,E2 -12547.932} C_VEL
LIN {X 0,Y 379.541,Z 646.965,A -85,B 0,C 180,E1 -12549.703,E2 -12549.703} C_VEL
LIN {X 0,Y 381.805,Z 634.462,A -85,B 0,C 180,E1 -12551.261,E2 -12551.261} C_VEL
LIN {X 0,Y 384.108,Z 620.287,A -85,B 0,C 180,E1 -12552.748,E2 -12552.748} C_VEL
LIN {X 0,Y 386.142,Z 606.6,A -85,B 0,C 180,E1 -12553.937,E2 -12553.937} C_VEL
LIN {X 0,Y 387.99,Z 592.601,A -85,B 0,C 180,E1 -12554.944,E2 -12554.944} C_VEL
LIN {X 0,Y 389.447,Z 577.758,A -85,B 0,C 180,E1 -12555.81,E2 -12555.81} C_VEL
LIN {X 0,Y 385.492,Z 564.818,A -85,B 0,C 180,E1 -12556.94,E2 -12556.94} C_VEL
LIN {X 0,Y 380.18,Z 551.607,A -85,B 0,C 180,E1 -12558.092,E2 -12558.092} C_VEL
LIN {X 0,Y 374.079,Z 538.773,A -85,B 0,C 180,E1 -12559.206,E2 -12559.206} C_VEL
LIN {X 0,Y 370.689,Z 532.255,A -85,B 0,C 180,E1 -12559.779,E2 -12559.779} C_VEL
LIN {X 0,Y 370.486,Z 531.437,A -85,B 0,C 180,E1 -12559.836,E2 -12559.836} C_VEL
LIN {X 0,Y 370.653,Z 526.943,A -85,B 0,C 180,E1 -12562.782,E2 -12562.782} C_VEL
LIN {X 0,Y 370.677,Z 523.118,A -85,B 0,C 180,E1 -12565.333,E2 -12565.333} C_VEL
LIN {X 0,Y 370.137,Z 519.318,A -85,B 0,C 180,E1 -12567.882,E2 -12567.882} C_VEL
LIN {X 0,Y 369.204,Z 514.031,A -85,B 0,C 180,E1 -12571.582,E2 -12571.582} C_VEL
LIN {X 0,Y 368.936,Z 512.844,A -85,B 0,C 180,E1 -12572.487,E2 -12572.487} C_VEL
LIN {X 0,Y 368.949,Z 512.84,A -85,B 0,C 180,E1 -12575.223,E2 -12575.223} C_VEL
LIN {X 0,Y 368.961,Z 512.837,A -85,B 0,C 180,E1 -12578.959,E2 -12578.959} C_VEL
LIN {X 0,Y 368.982,Z 512.838,A -85,B 0,C 180,E1 -12582.256,E2 -12582.256} C_VEL
LIN {X 0,Y 369.028,Z 512.825,A -85,B 0,C 180,E1 -12586.226,E2 -12586.226} C_VEL
LIN {X 0,Y 369.062,Z 512.827,A -85,B 0,C 180,E1 -12590.131,E2 -12590.131} C_VEL
LIN {X 0,Y 369.178,Z 512.805,A -85,B 0,C 180,E1 -12592.342,E2 -12592.342} C_VEL
LIN {X 0,Y 369.142,Z 512.812,A -85,B 0,C 180,E1 -12594.537,E2 -12594.537} C_VEL
LIN {X 0,Y 369.309,Z 512.79,A -85,B 0,C 180,E1 -12597.818,E2 -12597.818} C_VEL
LIN {X 0,Y 369.449,Z 512.779,A -85,B 0,C 180,E1 -12600,E2 -12600} C_VEL
LIN {X 0,Y 369.309,Z 512.787,A -85,B 0,C 180,E1 -12602.181,E2 -12602.181} C_VEL
LIN {X 0,Y 369.197,Z 512.806,A -85,B 0,C 180,E1 -12606.558,E2 -12606.558} C_VEL
LIN {X 0,Y 369.128,Z 512.807,A -85,B 0,C 180,E1 -12608.761,E2 -12608.761} C_VEL
LIN {X 0,Y 369.003,Z 512.823,A -85,B 0,C 180,E1 -12612.093,E2 -12612.093} C_VEL
LIN {X 0,Y 368.987,Z 512.825,A -85,B 0,C 180,E1 -12615.465,E2 -12615.465} C_VEL
LIN {X 0,Y 368.982,Z 512.804,A -85,B 0,C 180,E1 -12618.892,E2 -12618.892} C_VEL
LIN {X 0,Y 368.966,Z 512.83,A -85,B 0,C 180,E1 -12622.392,E2 -12622.392} C_VEL
LIN {X 0,Y 368.989,Z 512.81,A -85,B 0,C 180,E1 -12625.98,E2 -12625.98} C_VEL
LIN {X 0,Y 368.957,Z 512.84,A -85,B 0,C 180,E1 -12628.814,E2 -12628.814} C_VEL
LIN {X 0,Y 368.89,Z 512.847,A -85,B 0,C 180,E1 -12632.238,E2 -12632.238} C_VEL
LIN {X 0,Y 368.942,Z 512.934,A -85,B 0,C 180,E1 -12635.384,E2 -12635.384} C_VEL
LIN {X 0,Y 371.037,Z 522.197,A -85,B 0,C 180,E1 -12639.429,E2 -12639.429} C_VEL
LIN {X 0,Y 372.725,Z 530.278,A -85,B 0,C 180,E1 -12642.75,E2 -12642.75} C_VEL
LIN {X 0,Y 374.722,Z 539.616,A -85,B 0,C 180,E1 -12646.414,E2 -12646.414} C_VEL
LIN {X 0,Y 375.575,Z 545.122,A -85,B 0,C 180,E1 -12648.46,E2 -12648.46} C_VEL
LIN {X 0,Y 374.884,Z 552.83,A -85,B 0,C 180,E1 -12651.097,E2 -12651.097} C_VEL
LIN {X 0,Y 373.772,Z 562.657,A -85,B 0,C 180,E1 -12654.348,E2 -12654.348} C_VEL
LIN {X 0,Y 373.193,Z 568.173,A -85,B 0,C 180,E1 -12656.142,E2 -12656.142} C_VEL
LIN {X 0,Y 374.412,Z 572.337,A -85,B 0,C 180,E1 -12656.379,E2 -12656.379} C_VEL
LIN {X 0,Y 379.858,Z 592.097,A -85,B 0,C 180,E1 -12657.528,E2 -12657.528} C_VEL
LIN {X 0,Y 383.46,Z 608.29,A -85,B 0,C 180,E1 -12658.568,E2 -12658.568} C_VEL
LIN {X 0,Y 386.367,Z 624.586,A -85,B 0,C 180,E1 -12659.753,E2 -12659.753} C_VEL
LIN {X 0,Y 384.535,Z 640.556,A -85,B 0,C 180,E1 -12660.733,E2 -12660.733} C_VEL
LIN {X 0,Y 382.416,Z 655.326,A -85,B 0,C 180,E1 -12661.848,E2 -12661.848} C_VEL
LIN {X 0,Y 380.194,Z 670.137,A -85,B 0,C 180,E1 -12663.221,E2 -12663.221} C_VEL
LIN {X 0,Y 378.06,Z 683.36,A -85,B 0,C 180,E1 -12664.689,E2 -12664.689} C_VEL
LIN {X 0,Y 375.877,Z 696.143,A -85,B 0,C 180,E1 -12666.373,E2 -12666.373} C_VEL
LIN {X 0,Y 373.878,Z 707.841,A -85,B 0,C 180,E1 -12668.209,E2 -12668.209} C_VEL
LIN {X 0,Y 372.134,Z 718.285,A -85,B 0,C 180,E1 -12670.128,E2 -12670.128} C_VEL
LIN {X 0,Y 370.633,Z 728.452,A -85,B 0,C 180,E1 -12672.34,E2 -12672.34} C_VEL
LIN {X 0,Y 369.394,Z 737.013,A -85,B 0,C 180,E1 -12674.554,E2 -12674.554} C_VEL
LIN {X 0,Y 368.598,Z 744.08,A -85,B 0,C 180,E1 -12676.775,E2 -12676.775} C_VEL
LIN {X 0,Y 368.021,Z 749.932,A -85,B 0,C 180,E1 -12678.992,E2 -12678.992} C_VEL
LIN {X 0,Y 367.737,Z 754.638,A -85,B 0,C 180,E1 -12681.207,E2 -12681.207} C_VEL
LIN {X 0,Y 367.682,Z 758.557,A -85,B 0,C 180,E1 -12683.688,E2 -12683.688} C_VEL
LIN {X 0,Y 367.525,Z 760.751,A -85,B 0,C 180,E1 -12685.614,E2 -12685.614} C_VEL
LIN {X 0,Y 367.671,Z 762.223,A -85,B 0,C 180,E1 -12687.81,E2 -12687.81} C_VEL
LIN {X 0,Y 367.647,Z 762.775,A -85,B 0,C 180,E1 -12690.001,E2 -12690.001} C_VEL
LIN {X 0,Y 367.717,Z 762.242,A -85,B 0,C 180,E1 -12692.192,E2 -12692.192} C_VEL
LIN {X 0,Y 367.562,Z 760.776,A -85,B 0,C 180,E1 -12694.388,E2 -12694.388} C_VEL
LIN {X 0,Y 367.688,Z 758.216,A -85,B 0,C 180,E1 -12696.587,E2 -12696.587} C_VEL
LIN {X 0,Y 367.751,Z 754.648,A -85,B 0,C 180,E1 -12698.795,E2 -12698.795} C_VEL
LIN {X 0,Y 368.039,Z 749.932,A -85,B 0,C 180,E1 -12701.01,E2 -12701.01} C_VEL
LIN {X 0,Y 368.623,Z 744.037,A -85,B 0,C 180,E1 -12703.227,E2 -12703.227} C_VEL
LIN {X 0,Y 369.43,Z 736.89,A -85,B 0,C 180,E1 -12705.447,E2 -12705.447} C_VEL
LIN {X 0,Y 370.64,Z 728.226,A -85,B 0,C 180,E1 -12707.662,E2 -12707.662} C_VEL
LIN {X 0,Y 371.931,Z 719.244,A -85,B 0,C 180,E1 -12709.598,E2 -12709.598} C_VEL
LIN {X 0,Y 373.593,Z 708.813,A -85,B 0,C 180,E1 -12711.521,E2 -12711.521} C_VEL
LIN {X 0,Y 375.544,Z 696.776,A -85,B 0,C 180,E1 -12713.401,E2 -12713.401} C_VEL
LIN {X 0,Y 377.796,Z 683.073,A -85,B 0,C 180,E1 -12715.185,E2 -12715.185} C_VEL
LIN {X 0,Y 379.681,Z 670.8,A -85,B 0,C 180,E1 -12716.524,E2 -12716.524} C_VEL
LIN {X 0,Y 381.657,Z 656.568,A -85,B 0,C 180,E1 -12717.839,E2 -12717.839} C_VEL
LIN {X 0,Y 383.548,Z 642.627,A -85,B 0,C 180,E1 -12718.901,E2 -12718.901} C_VEL
LIN {X 0,Y 386.034,Z 624.028,A -85,B 0,C 180,E1 -12720.215,E2 -12720.215} C_VEL
LIN {X 0,Y 384.352,Z 610.064,A -85,B 0,C 180,E1 -12721.456,E2 -12721.456} C_VEL
LIN {X 0,Y 382.848,Z 592.163,A -85,B 0,C 180,E1 -12722.881,E2 -12722.881} C_VEL
LIN {X 0,Y 380.449,Z 578.104,A -85,B 0,C 180,E1 -12724.106,E2 -12724.106} C_VEL
LIN {X 0,Y 377.697,Z 567.278,A -85,B 0,C 180,E1 -12725.204,E2 -12725.204} C_VEL
LIN {X 0,Y 376.607,Z 563.103,A -85,B 0,C 180,E1 -12725.657,E2 -12725.657} C_VEL
LIN {X 0,Y 375.18,Z 557.853,A -85,B 0,C 180,E1 -12726.258,E2 -12726.258} C_VEL
LIN {X 0,Y 373.392,Z 552.581,A -85,B 0,C 180,E1 -12726.988,E2 -12726.988} C_VEL
LIN {X 0,Y 373.111,Z 550.545,A -85,B 0,C 180,E1 -12727.238,E2 -12727.238} C_VEL
LIN {X 0,Y 374.136,Z 542.091,A -85,B 0,C 180,E1 -12730.397,E2 -12730.397} C_VEL
LIN {X 0,Y 374.189,Z 538.656,A -85,B 0,C 180,E1 -12731.852,E2 -12731.852} C_VEL
LIN {X 0,Y 373.509,Z 533.622,A -85,B 0,C 180,E1 -12734.356,E2 -12734.356} C_VEL
LIN {X 0,Y 372.847,Z 529.992,A -85,B 0,C 180,E1 -12736.528,E2 -12736.528} C_VEL
LIN {X 0,Y 372.046,Z 526.622,A -85,B 0,C 180,E1 -12739.079,E2 -12739.079} C_VEL
LIN {X 0,Y 371.53,Z 524.313,A -85,B 0,C 180,E1 -12741.374,E2 -12741.374} C_VEL
LIN {X 0,Y 371.265,Z 523.046,A -85,B 0,C 180,E1 -12743.177,E2 -12743.177} C_VEL
LIN {X 0,Y 372.857,Z 525.318,A -85,B 0,C 180,E1 -12743.897,E2 -12743.897} C_VEL
LIN {X 0,Y 374.769,Z 526.624,A -85,B 0,C 180,E1 -12744.546,E2 -12744.546} C_VEL
LIN {X 0,Y 376.864,Z 529.064,A -85,B 0,C 180,E1 -12745.267,E2 -12745.267} C_VEL
LIN {X 0,Y 378.081,Z 530.226,A -85,B 0,C 180,E1 -12745.637,E2 -12745.637} C_VEL
LIN {X 0,Y 382.177,Z 535.266,A -85,B 0,C 180,E1 -12746.868,E2 -12746.868} C_VEL
LIN {X 0,Y 385.429,Z 540.024,A -85,B 0,C 180,E1 -12747.815,E2 -12747.815} C_VEL
LIN {X 0,Y 388.539,Z 547.458,A -85,B 0,C 180,E1 -12748.897,E2 -12748.897} C_VEL
LIN {X 0,Y 390.3,Z 552.725,A -85,B 0,C 180,E1 -12749.574,E2 -12749.574} C_VEL
LIN {X 0,Y 390.367,Z 554.418,A -85,B 0,C 180,E1 -12749.729,E2 -12749.729} C_VEL
LIN {X 0,Y 388.05,Z 570.451,A -85,B 0,C 180,E1 -12750.874,E2 -12750.874} C_VEL
LIN {X 0,Y 385.972,Z 583.992,A -85,B 0,C 180,E1 -12752.039,E2 -12752.039} C_VEL
LIN {X 0,Y 383.452,Z 599.268,A -85,B 0,C 180,E1 -12753.612,E2 -12753.612} C_VEL
LIN {X 0,Y 380.696,Z 614.196,A -85,B 0,C 180,E1 -12755.458,E2 -12755.458} C_VEL
LIN {X 0,Y 378.689,Z 625.112,A -85,B 0,C 180,E1 -12757.063,E2 -12757.063} C_VEL
LIN {X 0,Y 376.636,Z 635.84,A -85,B 0,C 180,E1 -12758.908,E2 -12758.908} C_VEL
LIN {X 0,Y 374.705,Z 645.377,A -85,B 0,C 180,E1 -12760.839,E2 -12760.839} C_VEL
LIN {X 0,Y 372.948,Z 654.439,A -85,B 0,C 180,E1 -12763.017,E2 -12763.017} C_VEL
LIN {X 0,Y 371.561,Z 661.953,A -85,B 0,C 180,E1 -12765.206,E2 -12765.206} C_VEL
LIN {X 0,Y 370.416,Z 668.172,A -85,B 0,C 180,E1 -12767.398,E2 -12767.398} C_VEL
LIN {X 0,Y 369.614,Z 673.069,A -85,B 0,C 180,E1 -12769.594,E2 -12769.594} C_VEL
LIN {X 0,Y 369.018,Z 677.264,A -85,B 0,C 180,E1 -12772.036,E2 -12772.036} C_VEL
LIN {X 0,Y 368.441,Z 680.255,A -85,B 0,C 180,E1 -12774.528,E2 -12774.528} C_VEL
LIN {X 0,Y 368.191,Z 681.784,A -85,B 0,C 180,E1 -12776.718,E2 -12776.718} C_VEL
LIN {X 0,Y 367.955,Z 682.339,A -85,B 0,C 180,E1 -12778.906,E2 -12778.906} C_VEL
LIN {X 0,Y 367.913,Z 681.955,A -85,B 0,C 180,E1 -12781.095,E2 -12781.095} C_VEL
LIN {X 0,Y 368.176,Z 680.518,A -85,B 0,C 180,E1 -12783.283,E2 -12783.283} C_VEL
LIN {X 0,Y 368.261,Z 678.186,A -85,B 0,C 180,E1 -12785.476,E2 -12785.476} C_VEL
LIN {X 0,Y 368.582,Z 673.76,A -85,B 0,C 180,E1 -12788.222,E2 -12788.222} C_VEL
LIN {X 0,Y 369.108,Z 667.608,A -85,B 0,C 180,E1 -12790.977,E2 -12790.977} C_VEL
LIN {X 0,Y 369.832,Z 661.302,A -85,B 0,C 180,E1 -12793.182,E2 -12793.182} C_VEL
LIN {X 0,Y 370.773,Z 653.664,A -85,B 0,C 180,E1 -12795.389,E2 -12795.389} C_VEL
LIN {X 0,Y 372.074,Z 644.508,A -85,B 0,C 180,E1 -12797.592,E2 -12797.592} C_VEL
LIN {X 0,Y 373.438,Z 635.124,A -85,B 0,C 180,E1 -12799.51,E2 -12799.51} C_VEL
LIN {X 0,Y 375.003,Z 624.007,A -85,B 0,C 180,E1 -12801.436,E2 -12801.436} C_VEL
LIN {X 0,Y 376.65,Z 612.958,A -85,B 0,C 180,E1 -12803.07,E2 -12803.07} C_VEL
LIN {X 0,Y 378.652,Z 599.217,A -85,B 0,C 180,E1 -12804.803,E2 -12804.803} C_VEL
LIN {X 0,Y 380.516,Z 585.032,A -85,B 0,C 180,E1 -12806.313,E2 -12806.313} C_VEL
LIN {X 0,Y 382.418,Z 570.642,A -85,B 0,C 180,E1 -12807.591,E2 -12807.591} C_VEL
LIN {X 0,Y 383.703,Z 558.05,A -85,B 0,C 180,E1 -12808.537,E2 -12808.537} C_VEL
LIN {X 0,Y 384.542,Z 550.192,A -85,B 0,C 180,E1 -12809.05,E2 -12809.05} C_VEL
LIN {X 0,Y 379.468,Z 536.957,A -85,B 0,C 180,E1 -12810.284,E2 -12810.284} C_VEL
LIN {X 0,Y 372.233,Z 520.715,A -85,B 0,C 180,E1 -12811.699,E2 -12811.699} C_VEL
LIN {X 0,Y 369.05,Z 513.467,A -85,B 0,C 180,E1 -12812.262,E2 -12812.262} C_VEL
LIN {X 0,Y 368.919,Z 512.845,A -85,B 0,C 180,E1 -12812.335,E2 -12812.335} C_VEL
LIN {X 0,Y 368.935,Z 512.842,A -85,B 0,C 180,E1 -12815.002,E2 -12815.002} C_VEL
LIN {X 0,Y 368.915,Z 512.845,A -85,B 0,C 180,E1 -12818.64,E2 -12818.64} C_VEL
LIN {X 0,Y 368.887,Z 512.849,A -85,B 0,C 180,E1 -12822.009,E2 -12822.009} C_VEL
LIN {X 0,Y 368.885,Z 512.847,A -85,B 0,C 180,E1 -12825.176,E2 -12825.176} C_VEL
LIN {X 0,Y 368.889,Z 512.847,A -85,B 0,C 180,E1 -12828.177,E2 -12828.177} C_VEL
LIN {X 0,Y 368.915,Z 512.846,A -85,B 0,C 180,E1 -12831.359,E2 -12831.359} C_VEL
LIN {X 0,Y 368.942,Z 512.842,A -85,B 0,C 180,E1 -12835.146,E2 -12835.146} C_VEL
LIN {X 0,Y 368.935,Z 512.846,A -85,B 0,C 180,E1 -12839.046,E2 -12839.046} C_VEL
LIN {X 0,Y 368.966,Z 512.905,A -85,B 0,C 180,E1 -12840.995,E2 -12840.995} C_VEL
LIN {X 0,Y 369.755,Z 517.81,A -85,B 0,C 180,E1 -12844.076,E2 -12844.076} C_VEL
LIN {X 0,Y 369.942,Z 521.696,A -85,B 0,C 180,E1 -12846.487,E2 -12846.487} C_VEL
LIN {X 0,Y 369.904,Z 525.509,A -85,B 0,C 180,E1 -12848.838,E2 -12848.838} C_VEL
LIN {X 0,Y 369.784,Z 530.138,A -85,B 0,C 180,E1 -12851.714,E2 -12851.714} C_VEL
LIN {X 0,Y 371.113,Z 533.526,A -85,B 0,C 180,E1 -12851.922,E2 -12851.922} C_VEL
LIN {X 0,Y 378.294,Z 550.957,A -85,B 0,C 180,E1 -12853.039,E2 -12853.039} C_VEL
LIN {X 0,Y 383.938,Z 566.631,A -85,B 0,C 180,E1 -12854.163,E2 -12854.163} C_VEL
LIN {X 0,Y 386.931,Z 576.301,A -85,B 0,C 180,E1 -12854.918,E2 -12854.918} C_VEL
LIN {X 0,Y 385.453,Z 592.384,A -85,B 0,C 180,E1 -12855.84,E2 -12855.84} C_VEL
LIN {X 0,Y 383.694,Z 607.131,A -85,B 0,C 180,E1 -12856.898,E2 -12856.898} C_VEL
LIN {X 0,Y 381.752,Z 621.657,A -85,B 0,C 180,E1 -12858.181,E2 -12858.181} C_VEL
LIN {X 0,Y 379.714,Z 635.09,A -85,B 0,C 180,E1 -12859.602,E2 -12859.602} C_VEL
LIN {X 0,Y 377.76,Z 647.545,A -85,B 0,C 180,E1 -12861.17,E2 -12861.17} C_VEL
LIN {X 0,Y 375.715,Z 659.543,A -85,B 0,C 180,E1 -12862.95,E2 -12862.95} C_VEL
LIN {X 0,Y 373.87,Z 670.407,A -85,B 0,C 180,E1 -12864.876,E2 -12864.876} C_VEL
LIN {X 0,Y 372.289,Z 679.404,A -85,B 0,C 180,E1 -12866.752,E2 -12866.752} C_VEL
LIN {X 0,Y 370.824,Z 688.191,A -85,B 0,C 180,E1 -12868.913,E2 -12868.913} C_VEL
LIN {X 0,Y 369.716,Z 695.546,A -85,B 0,C 180,E1 -12871.088,E2 -12871.088} C_VEL
LIN {X 0,Y 368.684,Z 702.963,A -85,B 0,C 180,E1 -12873.824,E2 -12873.824} C_VEL
LIN {X 0,Y 368.09,Z 708.611,A -85,B 0,C 180,E1 -12876.577,E2 -12876.577} C_VEL
LIN {X 0,Y 367.702,Z 711.927,A -85,B 0,C 180,E1 -12878.794,E2 -12878.794} C_VEL
LIN {X 0,Y 367.5,Z 714.317,A -85,B 0,C 180,E1 -12881.024,E2 -12881.024} C_VEL
LIN {X 0,Y 367.413,Z 715.662,A -85,B 0,C 180,E1 -12883.269,E2 -12883.269} C_VEL
LIN {X 0,Y 367.345,Z 716.077,A -85,B 0,C 180,E1 -12885.535,E2 -12885.535} C_VEL
LIN {X 0,Y 367.433,Z 715.474,A -85,B 0,C 180,E1 -12887.819,E2 -12887.819} C_VEL
LIN {X 0,Y 367.423,Z 715.134,A -85,B 0,C 180,E1 -12888.382,E2 -12888.382} C_VEL
LIN {X 0,Y 366.797,Z 714.62,A -85,B 0,C 180,E1 -12889.295,E2 -12889.295} C_VEL
LIN {X 0,Y 364.084,Z 713.52,A -85,B 0,C 180,E1 -12890.781,E2 -12890.781} C_VEL
LIN {X 0,Y 361.858,Z 712.383,A -85,B 0,C 180,E1 -12891.976,E2 -12891.976} C_VEL
LIN {X 0,Y 361.006,Z 711.257,A -85,B 0,C 180,E1 -12892.889,E2 -12892.889} C_VEL
LIN {X 0,Y 360.991,Z 710.801,A -85,B 0,C 180,E1 -12893.195,E2 -12893.195} C_VEL
LIN {X 0,Y 361.547,Z 707.228,A -85,B 0,C 180,E1 -12895.317,E2 -12895.317} C_VEL
LIN {X 0,Y 362.379,Z 701.941,A -85,B 0,C 180,E1 -12897.738,E2 -12897.738} C_VEL
LIN {X 0,Y 363.497,Z 695.289,A -85,B 0,C 180,E1 -12900.177,E2 -12900.177} C_VEL
LIN {X 0,Y 364.854,Z 688.464,A -85,B 0,C 180,E1 -12902.242,E2 -12902.242} C_VEL
LIN {X 0,Y 366.621,Z 679.553,A -85,B 0,C 180,E1 -12904.482,E2 -12904.482} C_VEL
LIN {X 0,Y 368.693,Z 669.63,A -85,B 0,C 180,E1 -12906.569,E2 -12906.569} C_VEL
LIN {X 0,Y 370.791,Z 659.569,A -85,B 0,C 180,E1 -12908.369,E2 -12908.369} C_VEL
LIN {X 0,Y 373.159,Z 647.704,A -85,B 0,C 180,E1 -12910.168,E2 -12910.168} C_VEL
LIN {X 0,Y 375.765,Z 634.143,A -85,B 0,C 180,E1 -12911.878,E2 -12911.878} C_VEL
LIN {X 0,Y 377.99,Z 620.884,A -85,B 0,C 180,E1 -12913.282,E2 -12913.282} C_VEL
LIN {X 0,Y 380.271,Z 605.745,A -85,B 0,C 180,E1 -12914.609,E2 -12914.609} C_VEL
LIN {X 0,Y 382.356,Z 590.299,A -85,B 0,C 180,E1 -12915.695,E2 -12915.695} C_VEL
LIN {X 0,Y 383.477,Z 580.194,A -85,B 0,C 180,E1 -12916.281,E2 -12916.281} C_VEL
LIN {X 0,Y 380.121,Z 568.632,A -85,B 0,C 180,E1 -12917.333,E2 -12917.333} C_VEL
LIN {X 0,Y 374.803,Z 554.959,A -85,B 0,C 180,E1 -12918.583,E2 -12918.583} C_VEL
LIN {X 0,Y 369.102,Z 542.778,A -85,B 0,C 180,E1 -12919.699,E2 -12919.699} C_VEL
LIN {X 0,Y 365.044,Z 535.229,A -85,B 0,C 180,E1 -12920.417,E2 -12920.417} C_VEL
LIN {X 0,Y 363.647,Z 531.874,A -85,B 0,C 180,E1 -12920.721,E2 -12920.721} C_VEL
LIN {X 0,Y 363.89,Z 526.628,A -85,B 0,C 180,E1 -12924.207,E2 -12924.207} C_VEL
LIN {X 0,Y 363.457,Z 522.267,A -85,B 0,C 180,E1 -12927.219,E2 -12927.219} C_VEL
LIN {X 0,Y 362.602,Z 517.243,A -85,B 0,C 180,E1 -12930.711,E2 -12930.711} C_VEL
LIN {X 0,Y 361.935,Z 513.712,A -85,B 0,C 180,E1 -12933.277,E2 -12933.277} C_VEL
LIN {X 0,Y 361.885,Z 513.719,A -85,B 0,C 180,E1 -12937.144,E2 -12937.144} C_VEL
LIN {X 0,Y 361.918,Z 513.714,A -85,B 0,C 180,E1 -12940.723,E2 -12940.723} C_VEL
LIN {X 0,Y 361.937,Z 513.711,A -85,B 0,C 180,E1 -12944.225,E2 -12944.225} C_VEL
LIN {X 0,Y 361.99,Z 513.702,A -85,B 0,C 180,E1 -12946.527,E2 -12946.527} C_VEL
LIN {X 0,Y 362.026,Z 513.701,A -85,B 0,C 180,E1 -12949.937,E2 -12949.937} C_VEL
LIN {X 0,Y 362.141,Z 513.681,A -85,B 0,C 180,E1 -12952.192,E2 -12952.192} C_VEL
LIN {X 0,Y 362.115,Z 513.688,A -85,B 0,C 180,E1 -12954.431,E2 -12954.431} C_VEL
LIN {X 0,Y 362.273,Z 513.666,A -85,B 0,C 180,E1 -12957.776,E2 -12957.776} C_VEL
LIN {X 0,Y 362.419,Z 513.654,A -85,B 0,C 180,E1 -12960,E2 -12960} C_VEL
LIN {X 0,Y 362.273,Z 513.663,A -85,B 0,C 180,E1 -12962.223,E2 -12962.223} C_VEL
LIN {X 0,Y 362.161,Z 513.684,A -85,B 0,C 180,E1 -12966.686,E2 -12966.686} C_VEL
LIN {X 0,Y 362.064,Z 513.686,A -85,B 0,C 180,E1 -12968.933,E2 -12968.933} C_VEL
LIN {X 0,Y 361.956,Z 513.7,A -85,B 0,C 180,E1 -12972.332,E2 -12972.332} C_VEL
LIN {X 0,Y 361.951,Z 513.71,A -85,B 0,C 180,E1 -12974.62,E2 -12974.62} C_VEL
LIN {X 0,Y 361.95,Z 513.67,A -85,B 0,C 180,E1 -12978.099,E2 -12978.099} C_VEL
LIN {X 0,Y 361.92,Z 513.716,A -85,B 0,C 180,E1 -12981.651,E2 -12981.651} C_VEL
LIN {X 0,Y 361.919,Z 513.68,A -85,B 0,C 180,E1 -12985.29,E2 -12985.29} C_VEL
LIN {X 0,Y 361.912,Z 513.719,A -85,B 0,C 180,E1 -12987.778,E2 -12987.778} C_VEL
LIN {X 0,Y 361.836,Z 513.726,A -85,B 0,C 180,E1 -12991.286,E2 -12991.286} C_VEL
LIN {X 0,Y 361.898,Z 513.784,A -85,B 0,C 180,E1 -12994.787,E2 -12994.787} C_VEL
LIN {X 0,Y 363.592,Z 521.427,A -85,B 0,C 180,E1 -12998.209,E2 -12998.209} C_VEL
LIN {X 0,Y 365.202,Z 528.847,A -85,B 0,C 180,E1 -13001.367,E2 -13001.367} C_VEL
LIN {X 0,Y 367.152,Z 538.04,A -85,B 0,C 180,E1 -13005.092,E2 -13005.092} C_VEL
LIN {X 0,Y 368.597,Z 545.701,A -85,B 0,C 180,E1 -13008.039,E2 -13008.039} C_VEL
LIN {X 0,Y 368.366,Z 550.522,A -85,B 0,C 180,E1 -13009.742,E2 -13009.742} C_VEL
LIN {X 0,Y 367.299,Z 559.898,A -85,B 0,C 180,E1 -13012.937,E2 -13012.937} C_VEL
LIN {X 0,Y 366.499,Z 567.259,A -85,B 0,C 180,E1 -13015.331,E2 -13015.331} C_VEL
LIN {X 0,Y 367.653,Z 571.155,A -85,B 0,C 180,E1 -13015.566,E2 -13015.566} C_VEL
LIN {X 0,Y 371.982,Z 585.931,A -85,B 0,C 180,E1 -13016.464,E2 -13016.464} C_VEL
LIN {X 0,Y 375.929,Z 602.599,A -85,B 0,C 180,E1 -13017.542,E2 -13017.542} C_VEL
LIN {X 0,Y 379.197,Z 620.365,A -85,B 0,C 180,E1 -13018.828,E2 -13018.828} C_VEL
LIN {X 0,Y 380.086,Z 626.795,A -85,B 0,C 180,E1 -13019.325,E2 -13019.325} C_VEL
LIN {X 0,Y 378.1,Z 642.665,A -85,B 0,C 180,E1 -13020.339,E2 -13020.339} C_VEL
LIN {X 0,Y 375.762,Z 658.034,A -85,B 0,C 180,E1 -13021.559,E2 -13021.559} C_VEL
LIN {X 0,Y 373.361,Z 672.654,A -85,B 0,C 180,E1 -13022.993,E2 -13022.993} C_VEL
LIN {X 0,Y 371.028,Z 686.414,A -85,B 0,C 180,E1 -13024.625,E2 -13024.625} C_VEL
LIN {X 0,Y 368.716,Z 699.09,A -85,B 0,C 180,E1 -13026.406,E2 -13026.406} C_VEL
LIN {X 0,Y 366.6,Z 710.741,A -85,B 0,C 180,E1 -13028.345,E2 -13028.345} C_VEL
LIN {X 0,Y 364.881,Z 720.726,A -85,B 0,C 180,E1 -13030.303,E2 -13030.303} C_VEL
LIN {X 0,Y 363.431,Z 730.373,A -85,B 0,C 180,E1 -13032.56,E2 -13032.56} C_VEL
LIN {X 0,Y 362.187,Z 738.492,A -85,B 0,C 180,E1 -13034.815,E2 -13034.815} C_VEL
LIN {X 0,Y 361.436,Z 745.292,A -85,B 0,C 180,E1 -13037.08,E2 -13037.08} C_VEL
LIN {X 0,Y 360.856,Z 750.796,A -85,B 0,C 180,E1 -13039.339,E2 -13039.339} C_VEL
LIN {X 0,Y 360.654,Z 754.216,A -85,B 0,C 180,E1 -13041.033,E2 -13041.033} C_VEL
LIN {X 0,Y 360.59,Z 758.332,A -85,B 0,C 180,E1 -13043.719,E2 -13043.719} C_VEL
LIN {X 0,Y 360.459,Z 760.313,A -85,B 0,C 180,E1 -13045.528,E2 -13045.528} C_VEL
LIN {X 0,Y 360.587,Z 761.779,A -85,B 0,C 180,E1 -13047.767,E2 -13047.767} C_VEL
LIN {X 0,Y 360.577,Z 762.324,A -85,B 0,C 180,E1 -13050.001,E2 -13050.001} C_VEL
LIN {X 0,Y 360.645,Z 761.786,A -85,B 0,C 180,E1 -13052.235,E2 -13052.235} C_VEL
LIN {X 0,Y 360.493,Z 760.31,A -85,B 0,C 180,E1 -13054.474,E2 -13054.474} C_VEL
LIN {X 0,Y 360.587,Z 757.742,A -85,B 0,C 180,E1 -13056.717,E2 -13056.717} C_VEL
LIN {X 0,Y 360.665,Z 754.162,A -85,B 0,C 180,E1 -13058.969,E2 -13058.969} C_VEL
LIN {X 0,Y 361.005,Z 749.437,A -85,B 0,C 180,E1 -13061.227,E2 -13061.227} C_VEL
LIN {X 0,Y 361.665,Z 742.939,A -85,B 0,C 180,E1 -13063.685,E2 -13063.685} C_VEL
LIN {X 0,Y 362.573,Z 735.302,A -85,B 0,C 180,E1 -13066.036,E2 -13066.036} C_VEL
LIN {X 0,Y 363.889,Z 726.513,A -85,B 0,C 180,E1 -13068.28,E2 -13068.28} C_VEL
LIN {X 0,Y 365.571,Z 715.879,A -85,B 0,C 180,E1 -13070.54,E2 -13070.54} C_VEL
LIN {X 0,Y 367.401,Z 704.872,A -85,B 0,C 180,E1 -13072.494,E2 -13072.494} C_VEL
LIN {X 0,Y 369.3,Z 693.875,A -85,B 0,C 180,E1 -13074.156,E2 -13074.156} C_VEL
LIN {X 0,Y 371.417,Z 681.15,A -85,B 0,C 180,E1 -13075.8,E2 -13075.8} C_VEL
LIN {X 0,Y 373.626,Z 667.368,A -85,B 0,C 180,E1 -13077.291,E2 -13077.291} C_VEL
LIN {X 0,Y 375.748,Z 652.956,A -85,B 0,C 180,E1 -13078.576,E2 -13078.576} C_VEL
LIN {X 0,Y 378.687,Z 633.714,A -85,B 0,C 180,E1 -13080.073,E2 -13080.073} C_VEL
LIN {X 0,Y 379.851,Z 626.324,A -85,B 0,C 180,E1 -13080.621,E2 -13080.621} C_VEL
LIN {X 0,Y 378.421,Z 611.12,A -85,B 0,C 180,E1 -13082.048,E2 -13082.048} C_VEL
LIN {X 0,Y 377.314,Z 594.314,A -85,B 0,C 180,E1 -13083.476,E2 -13083.476} C_VEL
LIN {X 0,Y 375.301,Z 581.074,A -85,B 0,C 180,E1 -13084.71,E2 -13084.71} C_VEL
LIN {X 0,Y 373.193,Z 571.439,A -85,B 0,C 180,E1 -13085.742,E2 -13085.742} C_VEL
LIN {X 0,Y 371.917,Z 566.525,A -85,B 0,C 180,E1 -13086.32,E2 -13086.32} C_VEL
LIN {X 0,Y 370.481,Z 560.997,A -85,B 0,C 180,E1 -13087.021,E2 -13087.021} C_VEL
LIN {X 0,Y 369.115,Z 555.687,A -85,B 0,C 180,E1 -13087.73,E2 -13087.73} C_VEL
LIN {X 0,Y 367.141,Z 549.935,A -85,B 0,C 180,E1 -13088.719,E2 -13088.719} C_VEL
LIN {X 0,Y 366.752,Z 547.44,A -85,B 0,C 180,E1 -13089.07,E2 -13089.07} C_VEL
LIN {X 0,Y 367.441,Z 542.269,A -85,B 0,C 180,E1 -13091.152,E2 -13091.152} C_VEL
LIN {X 0,Y 366.975,Z 537.217,A -85,B 0,C 180,E1 -13093.587,E2 -13093.587} C_VEL
LIN {X 0,Y 366.185,Z 532.602,A -85,B 0,C 180,E1 -13096.297,E2 -13096.297} C_VEL
LIN {X 0,Y 365.335,Z 528.849,A -85,B 0,C 180,E1 -13099.152,E2 -13099.152} C_VEL
LIN {X 0,Y 364.915,Z 526.945,A -85,B 0,C 180,E1 -13101.178,E2 -13101.178} C_VEL
LIN {X 0,Y 366.464,Z 528.871,A -85,B 0,C 180,E1 -13102.144,E2 -13102.144} C_VEL
LIN {X 0,Y 368.642,Z 529.926,A -85,B 0,C 180,E1 -13103.067,E2 -13103.067} C_VEL
LIN {X 0,Y 369.686,Z 531.381,A -85,B 0,C 180,E1 -13103.564,E2 -13103.564} C_VEL
LIN {X 0,Y 371.841,Z 533.11,A -85,B 0,C 180,E1 -13104.364,E2 -13104.364} C_VEL
LIN {X 0,Y 376.325,Z 538.284,A -85,B 0,C 180,E1 -13105.927,E2 -13105.927} C_VEL
LIN {X 0,Y 380.227,Z 543.672,A -85,B 0,C 180,E1 -13107.188,E2 -13107.188} C_VEL
LIN {X 0,Y 382.008,Z 547.286,A -85,B 0,C 180,E1 -13107.811,E2 -13107.811} C_VEL
LIN {X 0,Y 384.987,Z 556.248,A -85,B 0,C 180,E1 -13109.093,E2 -13109.093} C_VEL
LIN {X 0,Y 382.525,Z 572.049,A -85,B 0,C 180,E1 -13110.261,E2 -13110.261} C_VEL
LIN {X 0,Y 380.048,Z 586.644,A -85,B 0,C 180,E1 -13111.564,E2 -13111.564} C_VEL
LIN {X 0,Y 377.623,Z 600.362,A -85,B 0,C 180,E1 -13113.023,E2 -13113.023} C_VEL
LIN {X 0,Y 374.918,Z 614.212,A -85,B 0,C 180,E1 -13114.758,E2 -13114.758} C_VEL
LIN {X 0,Y 372.377,Z 626.847,A -85,B 0,C 180,E1 -13116.651,E2 -13116.651} C_VEL
LIN {X 0,Y 370.062,Z 638.008,A -85,B 0,C 180,E1 -13118.638,E2 -13118.638} C_VEL
LIN {X 0,Y 367.912,Z 648.065,A -85,B 0,C 180,E1 -13120.761,E2 -13120.761} C_VEL
LIN {X 0,Y 366.061,Z 656.767,A -85,B 0,C 180,E1 -13122.976,E2 -13122.976} C_VEL
LIN {X 0,Y 364.794,Z 663.193,A -85,B 0,C 180,E1 -13124.925,E2 -13124.925} C_VEL
LIN {X 0,Y 363.564,Z 669.315,A -85,B 0,C 180,E1 -13127.156,E2 -13127.156} C_VEL
LIN {X 0,Y 362.7,Z 674.173,A -85,B 0,C 180,E1 -13129.393,E2 -13129.393} C_VEL
LIN {X 0,Y 362.059,Z 678.287,A -85,B 0,C 180,E1 -13131.881,E2 -13131.881} C_VEL
LIN {X 0,Y 361.434,Z 681.212,A -85,B 0,C 180,E1 -13134.421,E2 -13134.421} C_VEL
LIN {X 0,Y 361.164,Z 682.704,A -85,B 0,C 180,E1 -13136.654,E2 -13136.654} C_VEL
LIN {X 0,Y 360.909,Z 683.207,A -85,B 0,C 180,E1 -13138.885,E2 -13138.885} C_VEL
LIN {X 0,Y 360.865,Z 682.772,A -85,B 0,C 180,E1 -13141.116,E2 -13141.116} C_VEL
LIN {X 0,Y 361.143,Z 681.265,A -85,B 0,C 180,E1 -13143.347,E2 -13143.347} C_VEL
LIN {X 0,Y 361.219,Z 678.877,A -85,B 0,C 180,E1 -13145.583,E2 -13145.583} C_VEL
LIN {X 0,Y 361.558,Z 674.372,A -85,B 0,C 180,E1 -13148.383,E2 -13148.383} C_VEL
LIN {X 0,Y 361.972,Z 669.498,A -85,B 0,C 180,E1 -13150.63,E2 -13150.63} C_VEL
LIN {X 0,Y 362.644,Z 663.453,A -85,B 0,C 180,E1 -13152.878,E2 -13152.878} C_VEL
LIN {X 0,Y 363.601,Z 656.119,A -85,B 0,C 180,E1 -13155.126,E2 -13155.126} C_VEL
LIN {X 0,Y 364.89,Z 647.272,A -85,B 0,C 180,E1 -13157.37,E2 -13157.37} C_VEL
LIN {X 0,Y 366.583,Z 635.976,A -85,B 0,C 180,E1 -13159.751,E2 -13159.751} C_VEL
LIN {X 0,Y 368.318,Z 624.07,A -85,B 0,C 180,E1 -13161.845,E2 -13161.845} C_VEL
LIN {X 0,Y 370.036,Z 612.889,A -85,B 0,C 180,E1 -13163.507,E2 -13163.507} C_VEL
LIN {X 0,Y 372.161,Z 598.775,A -85,B 0,C 180,E1 -13165.294,E2 -13165.294} C_VEL
LIN {X 0,Y 374.061,Z 584.631,A -85,B 0,C 180,E1 -13166.803,E2 -13166.803} C_VEL
LIN {X 0,Y 376.013,Z 570.313,A -85,B 0,C 180,E1 -13168.077,E2 -13168.077} C_VEL
LIN {X 0,Y 377.247,Z 558.561,A -85,B 0,C 180,E1 -13168.972,E2 -13168.972} C_VEL
LIN {X 0,Y 377.892,Z 553.057,A -85,B 0,C 180,E1 -13169.344,E2 -13169.344} C_VEL
LIN {X 0,Y 377.522,Z 550.862,A -85,B 0,C 180,E1 -13169.526,E2 -13169.526} C_VEL
LIN {X 0,Y 372.31,Z 537.628,A -85,B 0,C 180,E1 -13170.806,E2 -13170.806} C_VEL
LIN {X 0,Y 364.547,Z 520.038,A -85,B 0,C 180,E1 -13172.357,E2 -13172.357} C_VEL
LIN {X 0,Y 362.009,Z 514.454,A -85,B 0,C 180,E1 -13172.811,E2 -13172.811} C_VEL
LIN {X 0,Y 361.867,Z 513.723,A -85,B 0,C 180,E1 -13172.89,E2 -13172.89} C_VEL
LIN {X 0,Y 361.874,Z 513.722,A -85,B 0,C 180,E1 -13175.637,E2 -13175.637} C_VEL
LIN {X 0,Y 361.876,Z 513.724,A -85,B 0,C 180,E1 -13179.027,E2 -13179.027} C_VEL
LIN {X 0,Y 361.841,Z 513.727,A -85,B 0,C 180,E1 -13182.829,E2 -13182.829} C_VEL
LIN {X 0,Y 361.824,Z 513.729,A -85,B 0,C 180,E1 -13185.946,E2 -13185.946} C_VEL
LIN {X 0,Y 361.842,Z 513.726,A -85,B 0,C 180,E1 -13189.244,E2 -13189.244} C_VEL
LIN {X 0,Y 361.87,Z 513.721,A -85,B 0,C 180,E1 -13192.777,E2 -13192.777} C_VEL
LIN {X 0,Y 361.86,Z 513.726,A -85,B 0,C 180,E1 -13195.719,E2 -13195.719} C_VEL
LIN {X 0,Y 361.881,Z 513.727,A -85,B 0,C 180,E1 -13199.672,E2 -13199.672} C_VEL
LIN {X 0,Y 361.9,Z 513.857,A -85,B 0,C 180,E1 -13200.58,E2 -13200.58} C_VEL
LIN {X 0,Y 362.728,Z 518.46,A -85,B 0,C 180,E1 -13203.535,E2 -13203.535} C_VEL
LIN {X 0,Y 362.983,Z 522.398,A -85,B 0,C 180,E1 -13206.008,E2 -13206.008} C_VEL
LIN {X 0,Y 362.981,Z 526.258,A -85,B 0,C 180,E1 -13208.414,E2 -13208.414} C_VEL
LIN {X 0,Y 362.853,Z 530.714,A -85,B 0,C 180,E1 -13211.093,E2 -13211.093} C_VEL
LIN {X 0,Y 364.116,Z 533.797,A -85,B 0,C 180,E1 -13211.283,E2 -13211.283} C_VEL
LIN {X 0,Y 371.344,Z 551.117,A -85,B 0,C 180,E1 -13212.436,E2 -13212.436} C_VEL
LIN {X 0,Y 377.078,Z 566.869,A -85,B 0,C 180,E1 -13213.597,E2 -13213.597} C_VEL
LIN {X 0,Y 380.374,Z 577.691,A -85,B 0,C 180,E1 -13214.466,E2 -13214.466} C_VEL
LIN {X 0,Y 380.293,Z 581.319,A -85,B 0,C 180,E1 -13214.678,E2 -13214.678} C_VEL
LIN {X 0,Y 378.76,Z 595.963,A -85,B 0,C 180,E1 -13215.583,E2 -13215.583} C_VEL
LIN {X 0,Y 376.93,Z 610.223,A -85,B 0,C 180,E1 -13216.659,E2 -13216.659} C_VEL
LIN {X 0,Y 374.959,Z 624.409,A -85,B 0,C 180,E1 -13217.963,E2 -13217.963} C_VEL
LIN {X 0,Y 372.667,Z 638.6,A -85,B 0,C 180,E1 -13219.541,E2 -13219.541} C_VEL
LIN {X 0,Y 370.59,Z 651.474,A -85,B 0,C 180,E1 -13221.273,E2 -13221.273} C_VEL
LIN {X 0,Y 368.49,Z 662.843,A -85,B 0,C 180,E1 -13223.073,E2 -13223.073} C_VEL
LIN {X 0,Y 366.636,Z 673.384,A -85,B 0,C 180,E1 -13225.05,E2 -13225.05} C_VEL
LIN {X 0,Y 364.816,Z 683.222,A -85,B 0,C 180,E1 -13227.238,E2 -13227.238} C_VEL
LIN {X 0,Y 363.446,Z 691.441,A -85,B 0,C 180,E1 -13229.445,E2 -13229.445} C_VEL
LIN {X 0,Y 362.362,Z 698.282,A -85,B 0,C 180,E1 -13231.666,E2 -13231.666} C_VEL
LIN {X 0,Y 361.603,Z 703.958,A -85,B 0,C 180,E1 -13233.899,E2 -13233.899} C_VEL
LIN {X 0,Y 361.092,Z 708.483,A -85,B 0,C 180,E1 -13236.144,E2 -13236.144} C_VEL
LIN {X 0,Y 360.768,Z 711.233,A -85,B 0,C 180,E1 -13237.836,E2 -13237.836} C_VEL
LIN {X 0,Y 360.46,Z 713.939,A -85,B 0,C 180,E1 -13240.105,E2 -13240.105} C_VEL
LIN {X 0,Y 360.379,Z 715.914,A -85,B 0,C 180,E1 -13242.815,E2 -13242.815} C_VEL
LIN {X 0,Y 360.252,Z 716.477,A -85,B 0,C 180,E1 -13244.69,E2 -13244.69} C_VEL
LIN {X 0,Y 360.304,Z 716.253,A -85,B 0,C 180,E1 -13247.1,E2 -13247.1} C_VEL
LIN {X 0,Y 360.39,Z 715.056,A -85,B 0,C 180,E1 -13249.359,E2 -13249.359} C_VEL
LIN {X 0,Y 360.693,Z 712.762,A -85,B 0,C 180,E1 -13251.727,E2 -13251.727} C_VEL
LIN {X 0,Y 360.991,Z 710.801,A -85,B 0,C 180,E1 -13253.195,E2 -13253.195} C_VEL
LIN {X 0,Y 360.553,Z 709.494,A -85,B 0,C 180,E1 -13254.105,E2 -13254.105} C_VEL
LIN {X 0,Y 358.13,Z 707.184,A -85,B 0,C 180,E1 -13255.594,E2 -13255.594} C_VEL
LIN {X 0,Y 356.115,Z 705.086,A -85,B 0,C 180,E1 -13256.786,E2 -13256.786} C_VEL
LIN {X 0,Y 355.41,Z 703.235,A -85,B 0,C 180,E1 -13257.688,E2 -13257.688} C_VEL
LIN {X 0,Y 355.442,Z 702.534,A -85,B 0,C 180,E1 -13257.987,E2 -13257.987} C_VEL
LIN {X 0,Y 356.502,Z 696.684,A -85,B 0,C 180,E1 -13260.221,E2 -13260.221} C_VEL
LIN {X 0,Y 358.197,Z 688.443,A -85,B 0,C 180,E1 -13262.773,E2 -13262.773} C_VEL
LIN {X 0,Y 360.347,Z 678.536,A -85,B 0,C 180,E1 -13265.263,E2 -13265.263} C_VEL
LIN {X 0,Y 362.548,Z 668.414,A -85,B 0,C 180,E1 -13267.364,E2 -13267.364} C_VEL
LIN {X 0,Y 365.081,Z 656.525,A -85,B 0,C 180,E1 -13269.438,E2 -13269.438} C_VEL
LIN {X 0,Y 367.705,Z 644.025,A -85,B 0,C 180,E1 -13271.252,E2 -13271.252} C_VEL
LIN {X 0,Y 370.304,Z 630.55,A -85,B 0,C 180,E1 -13272.891,E2 -13272.891} C_VEL
LIN {X 0,Y 372.657,Z 617.211,A -85,B 0,C 180,E1 -13274.248,E2 -13274.248} C_VEL
LIN {X 0,Y 375.031,Z 601.616,A -85,B 0,C 180,E1 -13275.551,E2 -13275.551} C_VEL
LIN {X 0,Y 377.145,Z 585.538,A -85,B 0,C 180,E1 -13276.613,E2 -13276.613} C_VEL
LIN {X 0,Y 377.483,Z 582.096,A -85,B 0,C 180,E1 -13276.809,E2 -13276.809} C_VEL
LIN {X 0,Y 374.342,Z 571.283,A -85,B 0,C 180,E1 -13277.841,E2 -13277.841} C_VEL
LIN {X 0,Y 369.051,Z 557.352,A -85,B 0,C 180,E1 -13279.177,E2 -13279.177} C_VEL
LIN {X 0,Y 362.603,Z 543.697,A -85,B 0,C 180,E1 -13280.499,E2 -13280.499} C_VEL
LIN {X 0,Y 358.268,Z 535.705,A -85,B 0,C 180,E1 -13281.302,E2 -13281.302} C_VEL
LIN {X 0,Y 356.849,Z 532.386,A -85,B 0,C 180,E1 -13281.61,E2 -13281.61} C_VEL
LIN {X 0,Y 357.012,Z 529.097,A -85,B 0,C 180,E1 -13283.812,E2 -13283.812} C_VEL
LIN {X 0,Y 356.789,Z 525.221,A -85,B 0,C 180,E1 -13286.527,E2 -13286.527} C_VEL
LIN {X 0,Y 356.189,Z 521.522,A -85,B 0,C 180,E1 -13289.135,E2 -13289.135} C_VEL
LIN {X 0,Y 355.237,Z 516.281,A -85,B 0,C 180,E1 -13292.932,E2 -13292.932} C_VEL
LIN {X 0,Y 354.891,Z 514.592,A -85,B 0,C 180,E1 -13294.329,E2 -13294.329} C_VEL
LIN {X 0,Y 354.831,Z 514.602,A -85,B 0,C 180,E1 -13297.893,E2 -13297.893} C_VEL
LIN {X 0,Y 354.914,Z 514.588,A -85,B 0,C 180,E1 -13301.89,E2 -13301.89} C_VEL
LIN {X 0,Y 354.933,Z 514.58,A -85,B 0,C 180,E1 -13305.98,E2 -13305.98} C_VEL
LIN {X 0,Y 354.973,Z 514.577,A -85,B 0,C 180,E1 -13309.735,E2 -13309.735} C_VEL
LIN {X 0,Y 355.104,Z 514.557,A -85,B 0,C 180,E1 -13312.036,E2 -13312.036} C_VEL
LIN {X 0,Y 355.088,Z 514.564,A -85,B 0,C 180,E1 -13314.32,E2 -13314.32} C_VEL
LIN {X 0,Y 355.237,Z 514.543,A -85,B 0,C 180,E1 -13317.732,E2 -13317.732} C_VEL
LIN {X 0,Y 355.389,Z 514.53,A -85,B 0,C 180,E1 -13319.999,E2 -13319.999} C_VEL
LIN {X 0,Y 355.236,Z 514.54,A -85,B 0,C 180,E1 -13322.267,E2 -13322.267} C_VEL
LIN {X 0,Y 355.127,Z 514.56,A -85,B 0,C 180,E1 -13326.819,E2 -13326.819} C_VEL
LIN {X 0,Y 355.006,Z 514.565,A -85,B 0,C 180,E1 -13329.112,E2 -13329.112} C_VEL
LIN {X 0,Y 354.915,Z 514.576,A -85,B 0,C 180,E1 -13332.581,E2 -13332.581} C_VEL
LIN {X 0,Y 354.879,Z 514.566,A -85,B 0,C 180,E1 -13336.096,E2 -13336.096} C_VEL
LIN {X 0,Y 354.899,Z 514.55,A -85,B 0,C 180,E1 -13338.472,E2 -13338.472} C_VEL
LIN {X 0,Y 354.88,Z 514.587,A -85,B 0,C 180,E1 -13342.103,E2 -13342.103} C_VEL
LIN {X 0,Y 354.889,Z 514.561,A -85,B 0,C 180,E1 -13345.828,E2 -13345.828} C_VEL
LIN {X 0,Y 354.844,Z 514.597,A -85,B 0,C 180,E1 -13349.679,E2 -13349.679} C_VEL
LIN {X 0,Y 354.796,Z 514.603,A -85,B 0,C 180,E1 -13353.703,E2 -13353.703} C_VEL
LIN {X 0,Y 354.823,Z 514.699,A -85,B 0,C 180,E1 -13354.195,E2 -13354.195} C_VEL
LIN {X 0,Y 356.697,Z 522.998,A -85,B 0,C 180,E1 -13357.993,E2 -13357.993} C_VEL
LIN {X 0,Y 358.251,Z 530.14,A -85,B 0,C 180,E1 -13361.085,E2 -13361.085} C_VEL
LIN {X 0,Y 360.064,Z 538.757,A -85,B 0,C 180,E1 -13364.641,E2 -13364.641} C_VEL
LIN {X 0,Y 361.573,Z 546.303,A -85,B 0,C 180,E1 -13367.613,E2 -13367.613} C_VEL
LIN {X 0,Y 361.678,Z 549.107,A -85,B 0,C 180,E1 -13368.651,E2 -13368.651} C_VEL
LIN {X 0,Y 360.792,Z 557.091,A -85,B 0,C 180,E1 -13371.442,E2 -13371.442} C_VEL
LIN {X 0,Y 359.751,Z 565.883,A -85,B 0,C 180,E1 -13374.45,E2 -13374.45} C_VEL
LIN {X 0,Y 360.889,Z 569.868,A -85,B 0,C 180,E1 -13374.705,E2 -13374.705} C_VEL
LIN {X 0,Y 365.188,Z 583.751,A -85,B 0,C 180,E1 -13375.609,E2 -13375.609} C_VEL
LIN {X 0,Y 369.394,Z 601.214,A -85,B 0,C 180,E1 -13376.776,E2 -13376.776} C_VEL
LIN {X 0,Y 372.325,Z 617.443,A -85,B 0,C 180,E1 -13377.959,E2 -13377.959} C_VEL
LIN {X 0,Y 373.88,Z 628.25,A -85,B 0,C 180,E1 -13378.834,E2 -13378.834} C_VEL
LIN {X 0,Y 371.654,Z 644.59,A -85,B 0,C 180,E1 -13379.928,E2 -13379.928} C_VEL
LIN {X 0,Y 369.412,Z 658.672,A -85,B 0,C 180,E1 -13381.085,E2 -13381.085} C_VEL
LIN {X 0,Y 367.021,Z 672.648,A -85,B 0,C 180,E1 -13382.488,E2 -13382.488} C_VEL
LIN {X 0,Y 364.728,Z 685.251,A -85,B 0,C 180,E1 -13384.002,E2 -13384.002} C_VEL
LIN {X 0,Y 362.417,Z 697.327,A -85,B 0,C 180,E1 -13385.702,E2 -13385.702} C_VEL
LIN {X 0,Y 360.217,Z 708.988,A -85,B 0,C 180,E1 -13387.64,E2 -13387.64} C_VEL
LIN {X 0,Y 358.093,Z 720.449,A -85,B 0,C 180,E1 -13389.914,E2 -13389.914} C_VEL
LIN {X 0,Y 356.529,Z 730.061,A -85,B 0,C 180,E1 -13392.211,E2 -13392.211} C_VEL
LIN {X 0,Y 355.227,Z 738.136,A -85,B 0,C 180,E1 -13394.51,E2 -13394.51} C_VEL
LIN {X 0,Y 354.418,Z 744.903,A -85,B 0,C 180,E1 -13396.82,E2 -13396.82} C_VEL
LIN {X 0,Y 353.791,Z 750.398,A -85,B 0,C 180,E1 -13399.124,E2 -13399.124} C_VEL
LIN {X 0,Y 353.586,Z 753.811,A -85,B 0,C 180,E1 -13400.852,E2 -13400.852} C_VEL
LIN {X 0,Y 353.506,Z 758.104,A -85,B 0,C 180,E1 -13403.739,E2 -13403.739} C_VEL
LIN {X 0,Y 353.394,Z 759.881,A -85,B 0,C 180,E1 -13405.439,E2 -13405.439} C_VEL
LIN {X 0,Y 353.489,Z 761.336,A -85,B 0,C 180,E1 -13407.722,E2 -13407.722} C_VEL
LIN {X 0,Y 353.509,Z 761.872,A -85,B 0,C 180,E1 -13410.001,E2 -13410.001} C_VEL
LIN {X 0,Y 353.556,Z 761.325,A -85,B 0,C 180,E1 -13412.28,E2 -13412.28} C_VEL
LIN {X 0,Y 353.426,Z 759.836,A -85,B 0,C 180,E1 -13414.563,E2 -13414.563} C_VEL
LIN {X 0,Y 353.503,Z 757.258,A -85,B 0,C 180,E1 -13416.852,E2 -13416.852} C_VEL
LIN {X 0,Y 353.596,Z 753.656,A -85,B 0,C 180,E1 -13419.15,E2 -13419.15} C_VEL
LIN {X 0,Y 353.949,Z 748.919,A -85,B 0,C 180,E1 -13421.454,E2 -13421.454} C_VEL
LIN {X 0,Y 354.609,Z 742.856,A -85,B 0,C 180,E1 -13423.802,E2 -13423.802} C_VEL
LIN {X 0,Y 355.649,Z 734.744,A -85,B 0,C 180,E1 -13426.356,E2 -13426.356} C_VEL
LIN {X 0,Y 356.821,Z 727.071,A -85,B 0,C 180,E1 -13428.37,E2 -13428.37} C_VEL
LIN {X 0,Y 358.543,Z 716.638,A -85,B 0,C 180,E1 -13430.661,E2 -13430.661} C_VEL
LIN {X 0,Y 360.411,Z 705.846,A -85,B 0,C 180,E1 -13432.652,E2 -13432.652} C_VEL
LIN {X 0,Y 362.693,Z 693.169,A -85,B 0,C 180,E1 -13434.621,E2 -13434.621} C_VEL
LIN {X 0,Y 364.918,Z 680.368,A -85,B 0,C 180,E1 -13436.294,E2 -13436.294} C_VEL
LIN {X 0,Y 367.001,Z 667.869,A -85,B 0,C 180,E1 -13437.671,E2 -13437.671} C_VEL
LIN {X 0,Y 369.051,Z 654.584,A -85,B 0,C 180,E1 -13438.899,E2 -13438.899} C_VEL
LIN {X 0,Y 373.393,Z 629.721,A -85,B 0,C 180,E1 -13440.983,E2 -13440.983} C_VEL
LIN {X 0,Y 373.538,Z 626.13,A -85,B 0,C 180,E1 -13441.3,E2 -13441.3} C_VEL
LIN {X 0,Y 372.612,Z 613.484,A -85,B 0,C 180,E1 -13442.554,E2 -13442.554} C_VEL
LIN {X 0,Y 371.809,Z 596.323,A -85,B 0,C 180,E1 -13444.101,E2 -13444.101} C_VEL
LIN {X 0,Y 370.287,Z 584.334,A -85,B 0,C 180,E1 -13445.301,E2 -13445.301} C_VEL
LIN {X 0,Y 368.038,Z 572.3,A -85,B 0,C 180,E1 -13446.677,E2 -13446.677} C_VEL
LIN {X 0,Y 366.231,Z 565.009,A -85,B 0,C 180,E1 -13447.662,E2 -13447.662} C_VEL
LIN {X 0,Y 364.89,Z 559.444,A -85,B 0,C 180,E1 -13448.486,E2 -13448.486} C_VEL
LIN {X 0,Y 363.382,Z 554.016,A -85,B 0,C 180,E1 -13449.424,E2 -13449.424} C_VEL
LIN {X 0,Y 362.936,Z 552.025,A -85,B 0,C 180,E1 -13449.768,E2 -13449.768} C_VEL
LIN {X 0,Y 360.942,Z 544.77,A -85,B 0,C 180,E1 -13451.379,E2 -13451.379} C_VEL
LIN {X 0,Y 360.574,Z 542.734,A -85,B 0,C 180,E1 -13451.88,E2 -13451.88} C_VEL
LIN {X 0,Y 359.911,Z 537.459,A -85,B 0,C 180,E1 -13454.667,E2 -13454.667} C_VEL
LIN {X 0,Y 359.317,Z 534.135,A -85,B 0,C 180,E1 -13456.798,E2 -13456.798} C_VEL
LIN {X 0,Y 358.965,Z 532.772,A -85,B 0,C 180,E1 -13457.891,E2 -13457.891} C_VEL
LIN {X 0,Y 360.691,Z 533.586,A -85,B 0,C 180,E1 -13459.985,E2 -13459.985} C_VEL
LIN {X 0,Y 362.192,Z 533.659,A -85,B 0,C 180,E1 -13460.912,E2 -13460.912} C_VEL
LIN {X 0,Y 364.418,Z 535.738,A -85,B 0,C 180,E1 -13462.253,E2 -13462.253} C_VEL
LIN {X 0,Y 365.766,Z 536.309,A -85,B 0,C 180,E1 -13462.847,E2 -13462.847} C_VEL
LIN {X 0,Y 370.151,Z 541.111,A -85,B 0,C 180,E1 -13464.73,E2 -13464.73} C_VEL
LIN {X 0,Y 373.384,Z 545.132,A -85,B 0,C 180,E1 -13465.914,E2 -13465.914} C_VEL
LIN {X 0,Y 376.709,Z 550.16,A -85,B 0,C 180,E1 -13467.092,E2 -13467.092} C_VEL
LIN {X 0,Y 379.505,Z 558.495,A -85,B 0,C 180,E1 -13468.416,E2 -13468.416} C_VEL
LIN {X 0,Y 379.082,Z 562.364,A -85,B 0,C 180,E1 -13468.728,E2 -13468.728} C_VEL
LIN {X 0,Y 376.535,Z 576.943,A -85,B 0,C 180,E1 -13469.893,E2 -13469.893} C_VEL
LIN {X 0,Y 373.73,Z 592.056,A -85,B 0,C 180,E1 -13471.346,E2 -13471.346} C_VEL
LIN {X 0,Y 370.782,Z 607.06,A -85,B 0,C 180,E1 -13473.08,E2 -13473.08} C_VEL
LIN {X 0,Y 368.336,Z 618.124,A -85,B 0,C 180,E1 -13474.577,E2 -13474.577} C_VEL
LIN {X 0,Y 365.705,Z 630.252,A -85,B 0,C 180,E1 -13476.499,E2 -13476.499} C_VEL
LIN {X 0,Y 363.066,Z 642.019,A -85,B 0,C 180,E1 -13478.728,E2 -13478.728} C_VEL
LIN {X 0,Y 360.843,Z 651.8,A -85,B 0,C 180,E1 -13480.96,E2 -13480.96} C_VEL
LIN {X 0,Y 359.204,Z 659.147,A -85,B 0,C 180,E1 -13482.934,E2 -13482.934} C_VEL
LIN {X 0,Y 357.649,Z 666.092,A -85,B 0,C 180,E1 -13485.2,E2 -13485.2} C_VEL
LIN {X 0,Y 356.446,Z 671.791,A -85,B 0,C 180,E1 -13487.474,E2 -13487.474} C_VEL
LIN {X 0,Y 355.55,Z 676.344,A -85,B 0,C 180,E1 -13489.753,E2 -13489.753} C_VEL
LIN {X 0,Y 355.005,Z 679.762,A -85,B 0,C 180,E1 -13492.035,E2 -13492.035} C_VEL
LIN {X 0,Y 354.447,Z 682.19,A -85,B 0,C 180,E1 -13494.311,E2 -13494.311} C_VEL
LIN {X 0,Y 354.138,Z 683.63,A -85,B 0,C 180,E1 -13496.587,E2 -13496.587} C_VEL
LIN {X 0,Y 353.864,Z 684.067,A -85,B 0,C 180,E1 -13498.862,E2 -13498.862} C_VEL
LIN {X 0,Y 353.819,Z 683.585,A -85,B 0,C 180,E1 -13501.139,E2 -13501.139} C_VEL
LIN {X 0,Y 354.109,Z 682.016,A -85,B 0,C 180,E1 -13503.414,E2 -13503.414} C_VEL
LIN {X 0,Y 354.164,Z 679.548,A -85,B 0,C 180,E1 -13505.695,E2 -13505.695} C_VEL
LIN {X 0,Y 354.465,Z 675.995,A -85,B 0,C 180,E1 -13507.978,E2 -13507.978} C_VEL
LIN {X 0,Y 354.871,Z 671.353,A -85,B 0,C 180,E1 -13510.268,E2 -13510.268} C_VEL
LIN {X 0,Y 355.453,Z 665.587,A -85,B 0,C 180,E1 -13512.562,E2 -13512.562} C_VEL
LIN {X 0,Y 356.539,Z 657.927,A -85,B 0,C 180,E1 -13515.009,E2 -13515.009} C_VEL
LIN {X 0,Y 357.86,Z 648.716,A -85,B 0,C 180,E1 -13517.428,E2 -13517.428} C_VEL
LIN {X 0,Y 359.448,Z 638.527,A -85,B 0,C 180,E1 -13519.653,E2 -13519.653} C_VEL
LIN {X 0,Y 361.106,Z 627.447,A -85,B 0,C 180,E1 -13521.703,E2 -13521.703} C_VEL
LIN {X 0,Y 363.143,Z 614.774,A -85,B 0,C 180,E1 -13523.678,E2 -13523.678} C_VEL
LIN {X 0,Y 365.229,Z 601.339,A -85,B 0,C 180,E1 -13525.444,E2 -13525.444} C_VEL
LIN {X 0,Y 367.27,Z 587.029,A -85,B 0,C 180,E1 -13527.032,E2 -13527.032} C_VEL
LIN {X 0,Y 369.347,Z 572.136,A -85,B 0,C 180,E1 -13528.406,E2 -13528.406} C_VEL
LIN {X 0,Y 370.713,Z 559.736,A -85,B 0,C 180,E1 -13529.374,E2 -13529.374} C_VEL
LIN {X 0,Y 371.358,Z 553.934,A -85,B 0,C 180,E1 -13529.78,E2 -13529.78} C_VEL
LIN {X 0,Y 365.358,Z 538.672,A -85,B 0,C 180,E1 -13531.291,E2 -13531.291} C_VEL
LIN {X 0,Y 357.482,Z 520.794,A -85,B 0,C 180,E1 -13532.925,E2 -13532.925} C_VEL
LIN {X 0,Y 354.939,Z 515.226,A -85,B 0,C 180,E1 -13533.397,E2 -13533.397} C_VEL
LIN {X 0,Y 354.836,Z 514.6,A -85,B 0,C 180,E1 -13533.478,E2 -13533.478} C_VEL
LIN {X 0,Y 354.807,Z 514.602,A -85,B 0,C 180,E1 -13536.459,E2 -13536.459} C_VEL
LIN {X 0,Y 354.83,Z 514.599,A -85,B 0,C 180,E1 -13539.424,E2 -13539.424} C_VEL
LIN {X 0,Y 354.793,Z 514.605,A -85,B 0,C 180,E1 -13542.867,E2 -13542.867} C_VEL
LIN {X 0,Y 354.773,Z 514.608,A -85,B 0,C 180,E1 -13546.104,E2 -13546.104} C_VEL
LIN {X 0,Y 354.794,Z 514.605,A -85,B 0,C 180,E1 -13549.179,E2 -13549.179} C_VEL
LIN {X 0,Y 354.813,Z 514.602,A -85,B 0,C 180,E1 -13552.402,E2 -13552.402} C_VEL
LIN {X 0,Y 354.818,Z 514.602,A -85,B 0,C 180,E1 -13554.94,E2 -13554.94} C_VEL
LIN {X 0,Y 354.799,Z 514.61,A -85,B 0,C 180,E1 -13558.405,E2 -13558.405} C_VEL
LIN {X 0,Y 354.89,Z 514.804,A -85,B 0,C 180,E1 -13560.16,E2 -13560.16} C_VEL
LIN {X 0,Y 355.693,Z 519.139,A -85,B 0,C 180,E1 -13562.97,E2 -13562.97} C_VEL
LIN {X 0,Y 356.031,Z 523.126,A -85,B 0,C 180,E1 -13565.509,E2 -13565.509} C_VEL
LIN {X 0,Y 355.963,Z 528.984,A -85,B 0,C 180,E1 -13569.182,E2 -13569.182} C_VEL
LIN {X 0,Y 355.898,Z 530.945,A -85,B 0,C 180,E1 -13570.422,E2 -13570.422} C_VEL
LIN {X 0,Y 357.105,Z 534.16,A -85,B 0,C 180,E1 -13570.622,E2 -13570.622} C_VEL
LIN {X 0,Y 363.868,Z 549.841,A -85,B 0,C 180,E1 -13571.703,E2 -13571.703} C_VEL
LIN {X 0,Y 369.885,Z 566.215,A -85,B 0,C 180,E1 -13572.935,E2 -13572.935} C_VEL
LIN {X 0,Y 374.08,Z 579.714,A -85,B 0,C 180,E1 -13574.058,E2 -13574.058} C_VEL
LIN {X 0,Y 372.635,Z 594.62,A -85,B 0,C 180,E1 -13574.972,E2 -13574.972} C_VEL
LIN {X 0,Y 370.852,Z 608.65,A -85,B 0,C 180,E1 -13576.017,E2 -13576.017} C_VEL
LIN {X 0,Y 368.753,Z 623.086,A -85,B 0,C 180,E1 -13577.338,E2 -13577.338} C_VEL
LIN {X 0,Y 366.569,Z 636.443,A -85,B 0,C 180,E1 -13578.806,E2 -13578.806} C_VEL
LIN {X 0,Y 364.303,Z 649.771,A -85,B 0,C 180,E1 -13580.561,E2 -13580.561} C_VEL
LIN {X 0,Y 362.13,Z 661.524,A -85,B 0,C 180,E1 -13582.396,E2 -13582.396} C_VEL
LIN {X 0,Y 360.151,Z 672.337,A -85,B 0,C 180,E1 -13584.4,E2 -13584.4} C_VEL
LIN {X 0,Y 358.244,Z 682.369,A -85,B 0,C 180,E1 -13586.625,E2 -13586.625} C_VEL
LIN {X 0,Y 356.702,Z 690.788,A -85,B 0,C 180,E1 -13588.87,E2 -13588.87} C_VEL
LIN {X 0,Y 355.545,Z 697.844,A -85,B 0,C 180,E1 -13591.131,E2 -13591.131} C_VEL
LIN {X 0,Y 354.641,Z 703.701,A -85,B 0,C 180,E1 -13593.407,E2 -13593.407} C_VEL
LIN {X 0,Y 354.074,Z 708.347,A -85,B 0,C 180,E1 -13595.694,E2 -13595.694} C_VEL
LIN {X 0,Y 353.666,Z 712.023,A -85,B 0,C 180,E1 -13597.995,E2 -13597.995} C_VEL
LIN {X 0,Y 353.359,Z 714.633,A -85,B 0,C 180,E1 -13600.31,E2 -13600.31} C_VEL
LIN {X 0,Y 353.294,Z 716.398,A -85,B 0,C 180,E1 -13602.901,E2 -13602.901} C_VEL
LIN {X 0,Y 353.168,Z 716.969,A -85,B 0,C 180,E1 -13604.991,E2 -13604.991} C_VEL
LIN {X 0,Y 353.233,Z 716.64,A -85,B 0,C 180,E1 -13607.363,E2 -13607.363} C_VEL
LIN {X 0,Y 353.362,Z 715.339,A -85,B 0,C 180,E1 -13609.76,E2 -13609.76} C_VEL
LIN {X 0,Y 353.715,Z 712.897,A -85,B 0,C 180,E1 -13612.178,E2 -13612.178} C_VEL
LIN {X 0,Y 354.272,Z 709.381,A -85,B 0,C 180,E1 -13614.618,E2 -13614.618} C_VEL
LIN {X 0,Y 355.102,Z 704.642,A -85,B 0,C 180,E1 -13617.076,E2 -13617.076} C_VEL
LIN {X 0,Y 355.442,Z 702.534,A -85,B 0,C 180,E1 -13617.987,E2 -13617.987} C_VEL
LIN {X 0,Y 355.157,Z 700.488,A -85,B 0,C 180,E1 -13618.878,E2 -13618.878} C_VEL
LIN {X 0,Y 351.133,Z 693.341,A -85,B 0,C 180,E1 -13621.805,E2 -13621.805} C_VEL
LIN {X 0,Y 351.089,Z 690.641,A -85,B 0,C 180,E1 -13622.667,E2 -13622.667} C_VEL
LIN {X 0,Y 352.973,Z 682.305,A -85,B 0,C 180,E1 -13624.918,E2 -13624.918} C_VEL
LIN {X 0,Y 355.224,Z 672.606,A -85,B 0,C 180,E1 -13627.114,E2 -13627.114} C_VEL
LIN {X 0,Y 357.874,Z 661.044,A -85,B 0,C 180,E1 -13629.294,E2 -13629.294} C_VEL
LIN {X 0,Y 360.498,Z 649.264,A -85,B 0,C 180,E1 -13631.142,E2 -13631.142} C_VEL
LIN {X 0,Y 362.907,Z 637.754,A -85,B 0,C 180,E1 -13632.67,E2 -13632.67} C_VEL
LIN {X 0,Y 365.581,Z 623.626,A -85,B 0,C 180,E1 -13634.259,E2 -13634.259} C_VEL
LIN {X 0,Y 367.957,Z 609.78,A -85,B 0,C 180,E1 -13635.548,E2 -13635.548} C_VEL
LIN {X 0,Y 370.248,Z 594.662,A -85,B 0,C 180,E1 -13636.686,E2 -13636.686} C_VEL
LIN {X 0,Y 371.457,Z 585.084,A -85,B 0,C 180,E1 -13637.294,E2 -13637.294} C_VEL
LIN {X 0,Y 370.994,Z 582.016,A -85,B 0,C 180,E1 -13637.556,E2 -13637.556} C_VEL
LIN {X 0,Y 367.019,Z 569.306,A -85,B 0,C 180,E1 -13638.833,E2 -13638.833} C_VEL
LIN {X 0,Y 361.36,Z 555.307,A -85,B 0,C 180,E1 -13640.238,E2 -13640.238} C_VEL
LIN {X 0,Y 355.857,Z 544.135,A -85,B 0,C 180,E1 -13641.393,E2 -13641.393} C_VEL
LIN {X 0,Y 351.756,Z 536.551,A -85,B 0,C 180,E1 -13642.192,E2 -13642.192} C_VEL
LIN {X 0,Y 350.244,Z 533.628,A -85,B 0,C 180,E1 -13642.491,E2 -13642.491} C_VEL
LIN {X 0,Y 350.074,Z 532.794,A -85,B 0,C 180,E1 -13642.605,E2 -13642.605} C_VEL
LIN {X 0,Y 350.096,Z 528.775,A -85,B 0,C 180,E1 -13645.389,E2 -13645.389} C_VEL
LIN {X 0,Y 349.556,Z 524.534,A -85,B 0,C 180,E1 -13648.483,E2 -13648.483} C_VEL
LIN {X 0,Y 348.584,Z 519.158,A -85,B 0,C 180,E1 -13652.372,E2 -13652.372} C_VEL
LIN {X 0,Y 347.822,Z 515.471,A -85,B 0,C 180,E1 -13655.21,E2 -13655.21} C_VEL
LIN {X 0,Y 347.822,Z 515.47,A -85,B 0,C 180,E1 -13658.672,E2 -13658.672} C_VEL
LIN {X 0,Y 347.857,Z 515.47,A -85,B 0,C 180,E1 -13662.358,E2 -13662.358} C_VEL
LIN {X 0,Y 347.888,Z 515.457,A -85,B 0,C 180,E1 -13665.97,E2 -13665.97} C_VEL
LIN {X 0,Y 347.923,Z 515.453,A -85,B 0,C 180,E1 -13669.525,E2 -13669.525} C_VEL
LIN {X 0,Y 348.064,Z 515.434,A -85,B 0,C 180,E1 -13671.874,E2 -13671.874} C_VEL
LIN {X 0,Y 348.063,Z 515.44,A -85,B 0,C 180,E1 -13674.205,E2 -13674.205} C_VEL
LIN {X 0,Y 348.199,Z 515.42,A -85,B 0,C 180,E1 -13677.686,E2 -13677.686} C_VEL
LIN {X 0,Y 348.358,Z 515.406,A -85,B 0,C 180,E1 -13679.999,E2 -13679.999} C_VEL
LIN {X 0,Y 348.198,Z 515.416,A -85,B 0,C 180,E1 -13682.313,E2 -13682.313} C_VEL
LIN {X 0,Y 348.095,Z 515.436,A -85,B 0,C 180,E1 -13686.957,E2 -13686.957} C_VEL
LIN {X 0,Y 347.958,Z 515.444,A -85,B 0,C 180,E1 -13689.298,E2 -13689.298} C_VEL
LIN {X 0,Y 347.883,Z 515.453,A -85,B 0,C 180,E1 -13692.839,E2 -13692.839} C_VEL
LIN {X 0,Y 347.828,Z 515.436,A -85,B 0,C 180,E1 -13696.431,E2 -13696.431} C_VEL
LIN {X 0,Y 347.852,Z 515.431,A -85,B 0,C 180,E1 -13698.86,E2 -13698.86} C_VEL
LIN {X 0,Y 347.829,Z 515.471,A -85,B 0,C 180,E1 -13701.657,E2 -13701.657} C_VEL
LIN {X 0,Y 347.81,Z 515.433,A -85,B 0,C 180,E1 -13705.108,E2 -13705.108} C_VEL
LIN {X 0,Y 347.802,Z 515.476,A -85,B 0,C 180,E1 -13707.694,E2 -13707.694} C_VEL
LIN {X 0,Y 347.754,Z 515.482,A -85,B 0,C 180,E1 -13710.347,E2 -13710.347} C_VEL
LIN {X 0,Y 347.786,Z 515.594,A -85,B 0,C 180,E1 -13713.599,E2 -13713.599} C_VEL
LIN {X 0,Y 349.47,Z 523.081,A -85,B 0,C 180,E1 -13717.107,E2 -13717.107} C_VEL
LIN {X 0,Y 351.142,Z 530.703,A -85,B 0,C 180,E1 -13720.489,E2 -13720.489} C_VEL
LIN {X 0,Y 352.987,Z 539.535,A -85,B 0,C 180,E1 -13724.215,E2 -13724.215} C_VEL
LIN {X 0,Y 354.7,Z 548.103,A -85,B 0,C 180,E1 -13727.651,E2 -13727.651} C_VEL
LIN {X 0,Y 354.514,Z 553.204,A -85,B 0,C 180,E1 -13729.517,E2 -13729.517} C_VEL
LIN {X 0,Y 353.369,Z 562.256,A -85,B 0,C 180,E1 -13732.706,E2 -13732.706} C_VEL
LIN {X 0,Y 353.062,Z 564.912,A -85,B 0,C 180,E1 -13733.548,E2 -13733.548} C_VEL
LIN {X 0,Y 354.309,Z 568.958,A -85,B 0,C 180,E1 -13733.823,E2 -13733.823} C_VEL
LIN {X 0,Y 359.588,Z 585.738,A -85,B 0,C 180,E1 -13734.986,E2 -13734.986} C_VEL
LIN {X 0,Y 363.401,Z 602.637,A -85,B 0,C 180,E1 -13736.16,E2 -13736.16} C_VEL
LIN {X 0,Y 366.254,Z 619.107,A -85,B 0,C 180,E1 -13737.429,E2 -13737.429} C_VEL
LIN {X 0,Y 367.707,Z 629.228,A -85,B 0,C 180,E1 -13738.285,E2 -13738.285} C_VEL
LIN {X 0,Y 365.543,Z 644.868,A -85,B 0,C 180,E1 -13739.372,E2 -13739.372} C_VEL
